(* CODESYS project 4D_Handling_Demo_Seti.project

Project tree, tasks and I/O mapping:
  Device : CPX-CEC-M1-V3, Festo AG & Co. KG, order no. 3472765, version 3.5.7.25
      unmapped channels: Rotary switch
    application Application
      libraries: Standard, * (System); CAA CiA 405, 3.5.7.0 (CAA Technical Workgroup); Festo_Motion_FHPP_3, 3.5.5.0 (Festo AG & Co. KG)
      task MainTask (cyclic, interval t#20ms, priority 20) calls Main_PRG
      program Main_PRG [ST]
      PO3_Axis/
        AxisX/
          program PrgAxisXCallPrg [ST]
      program Motion_PRG [ST]
      program FHPP [CFC]
      global variables Global
      visualisation Visualization
    PLC_Diagnosis : PLC-Diagnosis, Festo AG & Co. KG, version 3.5.4.1
    CPX_System : CPX_System, Festo AG & Co. KG, order no. 3472765, version 1.200
      _8DI_8DO : 8DI/8DO, Festo AG & Co. KG, order no. 526257, version 1.200
          unmapped channels: Input 0, Output 0
      _8DI_8DO_1 : 8DI/8DO, Festo AG & Co. KG, order no. 526257, version 1.200
          settings:  = 0;  = 1;  = 1;  = 1;  = 1;  = 0;  = 1;  = 1;  = 0;  = 0;  = 0;  = 0;  = 0;  = 0;  = 0;  = 0;  = 0;  = 0;  = 0;  = 0;  = 0;  = 0;  = 0;  = 0;  = 0;  = 0;  = 0;  = 0;  = 0;  = 0;  = 0;  = 0;  = 0;  = 0;  = 0;  = 0;  = 0;  = 0;  = 0;  = 0;
             = 0;  = 0;  = 0;  = 0;  = 0;  = 0;  = 0;  = 0;  = 0;  = 0;  = 0;  = 0;  = 0;  = 0;  = 0;  = 0;  = 0;  = 0;  = 0;  = 0;  = 0;  = 0;  = 0;  = 0;  = 0;  = 0;  = 0;  = 0;  = 0;  = 0;  = 0;  = 0;  = 0;  = 0;  = 0;  = 0;  = 0;  = 0;  = 0;  = 0;
             = 576751027668385792;  = 'PI%i.0.0.1=1';  = 'PI%i.0.1.1=1';  = 'PI%i.0.2.1=1';  = 'PI%i.1.0.1=1';  = 'PI%i.1.1.1=0';  = 'PI%i.1.4.2=1';  = 'PI%i.1.6.2=1';  = 'PI%i.6.0.1=0';  = 'PI%i.6.1.1=0';  = 'PI%i.6.2.1=0';  = 'PI%i.6.3.1=0';  = 'PI%i.6.4.1=0';  = 'PI%i.6.5.1=0';  = 'PI%i.6.6.1=0';  = 'PI%i.6.7.1=0';  = dd1ef60a;  = 6
          unmapped channels: Input 0, Output 0
      CEC_M1_V3 : CEC-M1-V3, Festo AG & Co. KG, order no. 3472765, version 1.200
          settings:  = 0;  = 196272706293248;  = 352692416;  = 16777215;  = 0;  = 13959209;  = 1f4c82b2;  = 5
    SoftMotion General Axis Pool
    CAN : CANbus, 3S - Smart Software Solutions GmbH, version 3.5.7.0
        settings: Baudrate = 1000
      CANopen : CANopen_Manager, 3S - Smart Software Solutions GmbH, version 3.5.7.20
          settings: Sync CycleTime in Microseconds = 8000; Synchronous Window Length = 0; Enable Heartbeat generation = FALSE; Factory Settings Default = FALSE; Expert Settings Default = TRUE; ConfigVersion = 50659584
        U3 : CMMP-AS-C5-3A-M0 (FHPP), Festo AG & Co. KG, order no. 1622902, version 0.262146.CMMP_AS_C5_3A_M0_FHPP.2.8
            settings: General Options.Reset Node = FALSE; NODEIDSAVED = 3; SDO Timeout = 1000000; PDO_Autoconfig = FALSE; EXPERTSETTINGS = TRUE; Emergency-General Parameters.Emergency COBID = 16#00000083; PDO 16#1400.COBID = 16#00000203; PDO 16#1401.COBID = 16#00000303; PDO 16#1402.COBID = 16#00000403; PDO 16#1403.COBID = 16#00000503; PDO 16#1800.COBID = 16#00000183; PDO 16#1800.Event Timer = 0; PDO 16#1801.COBID = 16#00000283; PDO 16#1801.Event Timer = 0; PDO 16#1802.COBID = 16#00000383; PDO 16#1802.Event Timer = 0; PDO 16#1803.COBID = 16#00000483; PDO 16#1803.Event Timer = 0; CCON.Subindex = 16#00; CPOS.Subindex = 16#00; REC_NR/CDIR.Subindex = 16#00; RES/DEM_VAL1/PARA1.Subindex = 16#00; RES/DEM_VAL2/PARA2.Subindex = 16#00; RES.Subindex = 16#00; SUBINDEX.Subindex = 16#00; REQCODE_PNU.Subindex = 16#00; PARAVAL.Subindex = 16#00; FHPP+_O_Byte01.Subindex = 16#00; FHPP+_O_Byte02.Subindex = 16#00; FHPP+_O_Byte03.Subindex = 16#00; FHPP+_O_Byte04.Subindex = 16#00; FHPP+_O_Byte05.Subindex = 16#00; FHPP+_O_Byte06.Subindex = 16#00; FHPP+_O_Byte07.Subindex = 16#00; FHPP+_O_Byte08.Subindex = 16#00; FHPP+_O_Byte09.Subindex = 16#00; FHPP+_O_Byte10.Subindex = 16#00; FHPP+_O_Byte11.Subindex = 16#00; FHPP+_O_Byte12.Subindex = 16#00; FHPP+_O_Byte13.Subindex = 16#00;
              FHPP+_O_Byte14.Subindex = 16#00; FHPP+_O_Byte15.Subindex = 16#00; FHPP+_O_Byte16.Subindex = 16#00; SCON.Subindex = 16#00; SPOS.Subindex = 16#00; REC_NR/SDIR.Subindex = 16#00; RSB/ACT_VAL1.Subindex = 16#00; ACT_POS/ACT_VAL2.Subindex = 16#00; RES.Subindex = 16#00; SUBINDEX.Subindex = 16#00; RESPCODE_PNU.Subindex = 16#00; PARAVAL.Subindex = 16#00; FHPP+_I_Byte01.Subindex = 16#00; FHPP+_I_Byte02.Subindex = 16#00; FHPP+_I_Byte03.Subindex = 16#00; FHPP+_I_Byte04.Subindex = 16#00; FHPP+_I_Byte05.Subindex = 16#00; FHPP+_I_Byte06.Subindex = 16#00; FHPP+_I_Byte07.Subindex = 16#00; FHPP+_I_Byte08.Subindex = 16#00; FHPP+_I_Byte09.Subindex = 16#00; FHPP+_I_Byte10.Subindex = 16#00; FHPP+_I_Byte11.Subindex = 16#00; FHPP+_I_Byte12.Subindex = 16#00; FHPP+_I_Byte13.Subindex = 16#00; FHPP+_I_Byte14.Subindex = 16#00; FHPP+_I_Byte15.Subindex = 16#00; FHPP+_I_Byte16.Subindex = 16#00; SDO List.Disable TIME.Index = 16#1012; SDO List.Disable TIME.Subindex = 16#00; SDO List.Disable TIME.Value = 16#00000100; SDO List.Disable TIME.Size = 32; SDO List.Disable TIME.AbortIfError = FALSE; SDO List.Disable TIME.JumpToLine = FALSE; SDO List.Disable TIME.Line = 0; SDO List.Set Guardtime.Index = 16#100C; SDO List.Set Guardtime.Subindex = 16#00; SDO List.Set Guardtime.Value = 16#00000000; SDO List.Set Guardtime.Size = 16; SDO List.Set Guardtime.AbortIfError = FALSE;
              SDO List.Set Guardtime.JumpToLine = FALSE; SDO List.Set Guardtime.Line = 0; SDO List.Set Lifetime.Index = 16#100D; SDO List.Set Lifetime.Subindex = 16#00; SDO List.Set Lifetime.Value = 16#00000000; SDO List.Set Lifetime.Size = 8; SDO List.Set Lifetime.AbortIfError = FALSE; SDO List.Set Lifetime.JumpToLine = FALSE; SDO List.Set Lifetime.Line = 0; SDO List.Disable Emcy CobID.Index = 16#1014; SDO List.Disable Emcy CobID.Subindex = 16#00; SDO List.Disable Emcy CobID.Value = 16#80000083; SDO List.Disable Emcy CobID.Size = 32; SDO List.Disable Emcy CobID.AbortIfError = FALSE; SDO List.Disable Emcy CobID.JumpToLine = FALSE; SDO List.Disable Emcy CobID.Line = 0; SDO List.Set Emcy CobID.Index = 16#1014; SDO List.Set Emcy CobID.Subindex = 16#00; SDO List.Set Emcy CobID.Value = 16#00000083; SDO List.Set Emcy CobID.Size = 32; SDO List.Set Emcy CobID.AbortIfError = FALSE; SDO List.Set Emcy CobID.JumpToLine = FALSE; SDO List.Set Emcy CobID.Line = 0; SDO List.Set Heartbeat Consumer.Index = 16#1016; SDO List.Set Heartbeat Consumer.Subindex = 16#01; SDO List.Set Heartbeat Consumer.Value = 0; SDO List.Set Heartbeat Consumer.Size = 32; SDO List.Set Heartbeat Consumer.AbortIfError = FALSE; SDO List.Set Heartbeat Consumer.JumpToLine = FALSE; SDO List.Set Heartbeat Consumer.Line = 0; SDO List.Set Heartbeat Producer.Index = 16#1017; SDO List.Set Heartbeat Producer.Subindex = 16#00; SDO List.Set Heartbeat Producer.Value = 16#00000000; SDO List.Set Heartbeat Producer.Size = 16; SDO List.Set Heartbeat Producer.AbortIfError = FALSE; SDO List.Set Heartbeat Producer.JumpToLine = FALSE; SDO List.Set Heartbeat Producer.Line = 0; SDO List.Disable PDO.Index = 16#1400; SDO List.Disable PDO.Subindex = 16#01; SDO List.Disable PDO.Value = 16#80000203;
              SDO List.Disable PDO.Size = 32; SDO List.Disable PDO.AbortIfError = FALSE; SDO List.Disable PDO.JumpToLine = FALSE; SDO List.Disable PDO.Line = 0; SDO List.Set transmission type.Index = 16#1400; SDO List.Set transmission type.Subindex = 16#02; SDO List.Set transmission type.Value = 16#FF; SDO List.Set transmission type.Size = 8; SDO List.Set transmission type.AbortIfError = FALSE; SDO List.Set transmission type.JumpToLine = FALSE; SDO List.Set transmission type.Line = 0; SDO List.Set and enable COB-ID.Index = 16#1400; SDO List.Set and enable COB-ID.Subindex = 16#01; SDO List.Set and enable COB-ID.Value = 16#00000203; SDO List.Set and enable COB-ID.Size = 32; SDO List.Set and enable COB-ID.AbortIfError = FALSE; SDO List.Set and enable COB-ID.JumpToLine = FALSE; SDO List.Set and enable COB-ID.Line = 0; SDO List.Disable PDO.Index = 16#1401; SDO List.Disable PDO.Subindex = 16#01; SDO List.Disable PDO.Value = 16#80000303; SDO List.Disable PDO.Size = 32; SDO List.Disable PDO.AbortIfError = FALSE; SDO List.Disable PDO.JumpToLine = FALSE; SDO List.Disable PDO.Line = 0; SDO List.Set transmission type.Index = 16#1401; SDO List.Set transmission type.Subindex = 16#02; SDO List.Set transmission type.Value = 16#FF; SDO List.Set transmission type.Size = 8; SDO List.Set transmission type.AbortIfError = FALSE; SDO List.Set transmission type.JumpToLine = FALSE; SDO List.Set transmission type.Line = 0; SDO List.Set and enable COB-ID.Index = 16#1401; SDO List.Set and enable COB-ID.Subindex = 16#01; SDO List.Set and enable COB-ID.Value = 16#00000303; SDO List.Set and enable COB-ID.Size = 32; SDO List.Set and enable COB-ID.AbortIfError = FALSE; SDO List.Set and enable COB-ID.JumpToLine = FALSE; SDO List.Set and enable COB-ID.Line = 0; SDO List.Disable PDO.Index = 16#1402;
              SDO List.Disable PDO.Subindex = 16#01; SDO List.Disable PDO.Value = 16#80000403; SDO List.Disable PDO.Size = 32; SDO List.Disable PDO.AbortIfError = FALSE; SDO List.Disable PDO.JumpToLine = FALSE; SDO List.Disable PDO.Line = 0; SDO List.Set transmission type.Index = 16#1402; SDO List.Set transmission type.Subindex = 16#02; SDO List.Set transmission type.Value = 16#FF; SDO List.Set transmission type.Size = 8; SDO List.Set transmission type.AbortIfError = FALSE; SDO List.Set transmission type.JumpToLine = FALSE; SDO List.Set transmission type.Line = 0; SDO List.Clear pdo mapping.Index = 16#1602; SDO List.Clear pdo mapping.Subindex = 16#00; SDO List.Clear pdo mapping.Value = 16#0; SDO List.Clear pdo mapping.Size = 8; SDO List.Clear pdo mapping.AbortIfError = FALSE; SDO List.Clear pdo mapping.JumpToLine = FALSE; SDO List.Clear pdo mapping.Line = 0; SDO List.Set Mapping.Index = 16#1602; SDO List.Set Mapping.Subindex = 16#01; SDO List.Set Mapping.Value = 16#31010008; SDO List.Set Mapping.Size = 32; SDO List.Set Mapping.AbortIfError = FALSE; SDO List.Set Mapping.JumpToLine = FALSE; SDO List.Set Mapping.Line = 0; SDO List.Set Mapping.Index = 16#1602; SDO List.Set Mapping.Subindex = 16#02; SDO List.Set Mapping.Value = 16#31020008; SDO List.Set Mapping.Size = 32; SDO List.Set Mapping.AbortIfError = FALSE; SDO List.Set Mapping.JumpToLine = FALSE; SDO List.Set Mapping.Line = 0; SDO List.Set Mapping.Index = 16#1602; SDO List.Set Mapping.Subindex = 16#03; SDO List.Set Mapping.Value = 16#31030008; SDO List.Set Mapping.Size = 32; SDO List.Set Mapping.AbortIfError = FALSE; SDO List.Set Mapping.JumpToLine = FALSE;
              SDO List.Set Mapping.Line = 0; SDO List.Set Mapping.Index = 16#1602; SDO List.Set Mapping.Subindex = 16#04; SDO List.Set Mapping.Value = 16#31040008; SDO List.Set Mapping.Size = 32; SDO List.Set Mapping.AbortIfError = FALSE; SDO List.Set Mapping.JumpToLine = FALSE; SDO List.Set Mapping.Line = 0; SDO List.Set Mapping.Index = 16#1602; SDO List.Set Mapping.Subindex = 16#05; SDO List.Set Mapping.Value = 16#31050008; SDO List.Set Mapping.Size = 32; SDO List.Set Mapping.AbortIfError = FALSE; SDO List.Set Mapping.JumpToLine = FALSE; SDO List.Set Mapping.Line = 0; SDO List.Set Mapping.Index = 16#1602; SDO List.Set Mapping.Subindex = 16#06; SDO List.Set Mapping.Value = 16#31060008; SDO List.Set Mapping.Size = 32; SDO List.Set Mapping.AbortIfError = FALSE; SDO List.Set Mapping.JumpToLine = FALSE; SDO List.Set Mapping.Line = 0; SDO List.Set Mapping.Index = 16#1602; SDO List.Set Mapping.Subindex = 16#07; SDO List.Set Mapping.Value = 16#31070008; SDO List.Set Mapping.Size = 32; SDO List.Set Mapping.AbortIfError = FALSE; SDO List.Set Mapping.JumpToLine = FALSE; SDO List.Set Mapping.Line = 0; SDO List.Set Mapping.Index = 16#1602; SDO List.Set Mapping.Subindex = 16#08; SDO List.Set Mapping.Value = 16#31080008; SDO List.Set Mapping.Size = 32; SDO List.Set Mapping.AbortIfError = FALSE; SDO List.Set Mapping.JumpToLine = FALSE; SDO List.Set Mapping.Line = 0; SDO List.Set number of mappings.Index = 16#1602; SDO List.Set number of mappings.Subindex = 16#00; SDO List.Set number of mappings.Value = 16#08; SDO List.Set number of mappings.Size = 8;
              SDO List.Set number of mappings.AbortIfError = FALSE; SDO List.Set number of mappings.JumpToLine = FALSE; SDO List.Set number of mappings.Line = 0; SDO List.Set and enable COB-ID.Index = 16#1402; SDO List.Set and enable COB-ID.Subindex = 16#01; SDO List.Set and enable COB-ID.Value = 16#00000403; SDO List.Set and enable COB-ID.Size = 32; SDO List.Set and enable COB-ID.AbortIfError = FALSE; SDO List.Set and enable COB-ID.JumpToLine = FALSE; SDO List.Set and enable COB-ID.Line = 0; SDO List.Disable PDO.Index = 16#1403; SDO List.Disable PDO.Subindex = 16#01; SDO List.Disable PDO.Value = 16#80000503; SDO List.Disable PDO.Size = 32; SDO List.Disable PDO.AbortIfError = FALSE; SDO List.Disable PDO.JumpToLine = FALSE; SDO List.Disable PDO.Line = 0; SDO List.Set transmission type.Index = 16#1403; SDO List.Set transmission type.Subindex = 16#02; SDO List.Set transmission type.Value = 16#FF; SDO List.Set transmission type.Size = 8; SDO List.Set transmission type.AbortIfError = FALSE; SDO List.Set transmission type.JumpToLine = FALSE; SDO List.Set transmission type.Line = 0; SDO List.Clear pdo mapping.Index = 16#1603; SDO List.Clear pdo mapping.Subindex = 16#00; SDO List.Clear pdo mapping.Value = 16#0; SDO List.Clear pdo mapping.Size = 8; SDO List.Clear pdo mapping.AbortIfError = FALSE; SDO List.Clear pdo mapping.JumpToLine = FALSE; SDO List.Clear pdo mapping.Line = 0; SDO List.Set Mapping.Index = 16#1603; SDO List.Set Mapping.Subindex = 16#01; SDO List.Set Mapping.Value = 16#31090008; SDO List.Set Mapping.Size = 32; SDO List.Set Mapping.AbortIfError = FALSE; SDO List.Set Mapping.JumpToLine = FALSE; SDO List.Set Mapping.Line = 0; SDO List.Set Mapping.Index = 16#1603; SDO List.Set Mapping.Subindex = 16#02;
              SDO List.Set Mapping.Value = 16#31100008; SDO List.Set Mapping.Size = 32; SDO List.Set Mapping.AbortIfError = FALSE; SDO List.Set Mapping.JumpToLine = FALSE; SDO List.Set Mapping.Line = 0; SDO List.Set Mapping.Index = 16#1603; SDO List.Set Mapping.Subindex = 16#03; SDO List.Set Mapping.Value = 16#31110008; SDO List.Set Mapping.Size = 32; SDO List.Set Mapping.AbortIfError = FALSE; SDO List.Set Mapping.JumpToLine = FALSE; SDO List.Set Mapping.Line = 0; SDO List.Set Mapping.Index = 16#1603; SDO List.Set Mapping.Subindex = 16#04; SDO List.Set Mapping.Value = 16#31120008; SDO List.Set Mapping.Size = 32; SDO List.Set Mapping.AbortIfError = FALSE; SDO List.Set Mapping.JumpToLine = FALSE; SDO List.Set Mapping.Line = 0; SDO List.Set Mapping.Index = 16#1603; SDO List.Set Mapping.Subindex = 16#05; SDO List.Set Mapping.Value = 16#31130008; SDO List.Set Mapping.Size = 32; SDO List.Set Mapping.AbortIfError = FALSE; SDO List.Set Mapping.JumpToLine = FALSE; SDO List.Set Mapping.Line = 0; SDO List.Set Mapping.Index = 16#1603; SDO List.Set Mapping.Subindex = 16#06; SDO List.Set Mapping.Value = 16#31140008; SDO List.Set Mapping.Size = 32; SDO List.Set Mapping.AbortIfError = FALSE; SDO List.Set Mapping.JumpToLine = FALSE; SDO List.Set Mapping.Line = 0; SDO List.Set Mapping.Index = 16#1603; SDO List.Set Mapping.Subindex = 16#07; SDO List.Set Mapping.Value = 16#31150008; SDO List.Set Mapping.Size = 32; SDO List.Set Mapping.AbortIfError = FALSE; SDO List.Set Mapping.JumpToLine = FALSE; SDO List.Set Mapping.Line = 0;
              SDO List.Set Mapping.Index = 16#1603; SDO List.Set Mapping.Subindex = 16#08; SDO List.Set Mapping.Value = 16#31160008; SDO List.Set Mapping.Size = 32; SDO List.Set Mapping.AbortIfError = FALSE; SDO List.Set Mapping.JumpToLine = FALSE; SDO List.Set Mapping.Line = 0; SDO List.Set number of mappings.Index = 16#1603; SDO List.Set number of mappings.Subindex = 16#00; SDO List.Set number of mappings.Value = 16#08; SDO List.Set number of mappings.Size = 8; SDO List.Set number of mappings.AbortIfError = FALSE; SDO List.Set number of mappings.JumpToLine = FALSE; SDO List.Set number of mappings.Line = 0; SDO List.Set and enable COB-ID.Index = 16#1403; SDO List.Set and enable COB-ID.Subindex = 16#01; SDO List.Set and enable COB-ID.Value = 16#00000503; SDO List.Set and enable COB-ID.Size = 32; SDO List.Set and enable COB-ID.AbortIfError = FALSE; SDO List.Set and enable COB-ID.JumpToLine = FALSE; SDO List.Set and enable COB-ID.Line = 0; SDO List.Disable PDO.Index = 16#1800; SDO List.Disable PDO.Subindex = 16#01; SDO List.Disable PDO.Value = 16#80000183; SDO List.Disable PDO.Size = 32; SDO List.Disable PDO.AbortIfError = FALSE; SDO List.Disable PDO.JumpToLine = FALSE; SDO List.Disable PDO.Line = 0; SDO List.Set transmission type.Index = 16#1800; SDO List.Set transmission type.Subindex = 16#02; SDO List.Set transmission type.Value = 16#FF; SDO List.Set transmission type.Size = 8; SDO List.Set transmission type.AbortIfError = FALSE; SDO List.Set transmission type.JumpToLine = FALSE; SDO List.Set transmission type.Line = 0; SDO List.Set inhibit time.Index = 16#1800; SDO List.Set inhibit time.Subindex = 16#03; SDO List.Set inhibit time.Value = 16#0000; SDO List.Set inhibit time.Size = 16; SDO List.Set inhibit time.AbortIfError = FALSE;
              SDO List.Set inhibit time.JumpToLine = FALSE; SDO List.Set inhibit time.Line = 0; SDO List.Set and enable COB-ID.Index = 16#1800; SDO List.Set and enable COB-ID.Subindex = 16#01; SDO List.Set and enable COB-ID.Value = 16#00000183; SDO List.Set and enable COB-ID.Size = 32; SDO List.Set and enable COB-ID.AbortIfError = FALSE; SDO List.Set and enable COB-ID.JumpToLine = FALSE; SDO List.Set and enable COB-ID.Line = 0; SDO List.Disable PDO.Index = 16#1801; SDO List.Disable PDO.Subindex = 16#01; SDO List.Disable PDO.Value = 16#80000283; SDO List.Disable PDO.Size = 32; SDO List.Disable PDO.AbortIfError = FALSE; SDO List.Disable PDO.JumpToLine = FALSE; SDO List.Disable PDO.Line = 0; SDO List.Set transmission type.Index = 16#1801; SDO List.Set transmission type.Subindex = 16#02; SDO List.Set transmission type.Value = 16#FF; SDO List.Set transmission type.Size = 8; SDO List.Set transmission type.AbortIfError = FALSE; SDO List.Set transmission type.JumpToLine = FALSE; SDO List.Set transmission type.Line = 0; SDO List.Set inhibit time.Index = 16#1801; SDO List.Set inhibit time.Subindex = 16#03; SDO List.Set inhibit time.Value = 16#0000; SDO List.Set inhibit time.Size = 16; SDO List.Set inhibit time.AbortIfError = FALSE; SDO List.Set inhibit time.JumpToLine = FALSE; SDO List.Set inhibit time.Line = 0; SDO List.Set and enable COB-ID.Index = 16#1801; SDO List.Set and enable COB-ID.Subindex = 16#01; SDO List.Set and enable COB-ID.Value = 16#00000283; SDO List.Set and enable COB-ID.Size = 32; SDO List.Set and enable COB-ID.AbortIfError = FALSE; SDO List.Set and enable COB-ID.JumpToLine = FALSE; SDO List.Set and enable COB-ID.Line = 0; SDO List.Disable PDO.Index = 16#1802; SDO List.Disable PDO.Subindex = 16#01; SDO List.Disable PDO.Value = 16#80000383;
              SDO List.Disable PDO.Size = 32; SDO List.Disable PDO.AbortIfError = FALSE; SDO List.Disable PDO.JumpToLine = FALSE; SDO List.Disable PDO.Line = 0; SDO List.Set transmission type.Index = 16#1802; SDO List.Set transmission type.Subindex = 16#02; SDO List.Set transmission type.Value = 16#FF; SDO List.Set transmission type.Size = 8; SDO List.Set transmission type.AbortIfError = FALSE; SDO List.Set transmission type.JumpToLine = FALSE; SDO List.Set transmission type.Line = 0; SDO List.Set inhibit time.Index = 16#1802; SDO List.Set inhibit time.Subindex = 16#03; SDO List.Set inhibit time.Value = 16#0000; SDO List.Set inhibit time.Size = 16; SDO List.Set inhibit time.AbortIfError = FALSE; SDO List.Set inhibit time.JumpToLine = FALSE; SDO List.Set inhibit time.Line = 0; SDO List.Clear pdo mapping.Index = 16#1A02; SDO List.Clear pdo mapping.Subindex = 16#00; SDO List.Clear pdo mapping.Value = 16#0; SDO List.Clear pdo mapping.Size = 8; SDO List.Clear pdo mapping.AbortIfError = FALSE; SDO List.Clear pdo mapping.JumpToLine = FALSE; SDO List.Clear pdo mapping.Line = 0; SDO List.Set Mapping.Index = 16#1A02; SDO List.Set Mapping.Subindex = 16#01; SDO List.Set Mapping.Value = 16#32010008; SDO List.Set Mapping.Size = 32; SDO List.Set Mapping.AbortIfError = FALSE; SDO List.Set Mapping.JumpToLine = FALSE; SDO List.Set Mapping.Line = 0; SDO List.Set Mapping.Index = 16#1A02; SDO List.Set Mapping.Subindex = 16#02; SDO List.Set Mapping.Value = 16#32020008; SDO List.Set Mapping.Size = 32; SDO List.Set Mapping.AbortIfError = FALSE; SDO List.Set Mapping.JumpToLine = FALSE; SDO List.Set Mapping.Line = 0; SDO List.Set Mapping.Index = 16#1A02;
              SDO List.Set Mapping.Subindex = 16#03; SDO List.Set Mapping.Value = 16#32030008; SDO List.Set Mapping.Size = 32; SDO List.Set Mapping.AbortIfError = FALSE; SDO List.Set Mapping.JumpToLine = FALSE; SDO List.Set Mapping.Line = 0; SDO List.Set Mapping.Index = 16#1A02; SDO List.Set Mapping.Subindex = 16#04; SDO List.Set Mapping.Value = 16#32040008; SDO List.Set Mapping.Size = 32; SDO List.Set Mapping.AbortIfError = FALSE; SDO List.Set Mapping.JumpToLine = FALSE; SDO List.Set Mapping.Line = 0; SDO List.Set Mapping.Index = 16#1A02; SDO List.Set Mapping.Subindex = 16#05; SDO List.Set Mapping.Value = 16#32050008; SDO List.Set Mapping.Size = 32; SDO List.Set Mapping.AbortIfError = FALSE; SDO List.Set Mapping.JumpToLine = FALSE; SDO List.Set Mapping.Line = 0; SDO List.Set Mapping.Index = 16#1A02; SDO List.Set Mapping.Subindex = 16#06; SDO List.Set Mapping.Value = 16#32060008; SDO List.Set Mapping.Size = 32; SDO List.Set Mapping.AbortIfError = FALSE; SDO List.Set Mapping.JumpToLine = FALSE; SDO List.Set Mapping.Line = 0; SDO List.Set Mapping.Index = 16#1A02; SDO List.Set Mapping.Subindex = 16#07; SDO List.Set Mapping.Value = 16#32070008; SDO List.Set Mapping.Size = 32; SDO List.Set Mapping.AbortIfError = FALSE; SDO List.Set Mapping.JumpToLine = FALSE; SDO List.Set Mapping.Line = 0; SDO List.Set Mapping.Index = 16#1A02; SDO List.Set Mapping.Subindex = 16#08; SDO List.Set Mapping.Value = 16#32080008; SDO List.Set Mapping.Size = 32; SDO List.Set Mapping.AbortIfError = FALSE; SDO List.Set Mapping.JumpToLine = FALSE;
              SDO List.Set Mapping.Line = 0; SDO List.Set number of mappings.Index = 16#1A02; SDO List.Set number of mappings.Subindex = 16#00; SDO List.Set number of mappings.Value = 16#08; SDO List.Set number of mappings.Size = 8; SDO List.Set number of mappings.AbortIfError = FALSE; SDO List.Set number of mappings.JumpToLine = FALSE; SDO List.Set number of mappings.Line = 0; SDO List.Set and enable COB-ID.Index = 16#1802; SDO List.Set and enable COB-ID.Subindex = 16#01; SDO List.Set and enable COB-ID.Value = 16#00000383; SDO List.Set and enable COB-ID.Size = 32; SDO List.Set and enable COB-ID.AbortIfError = FALSE; SDO List.Set and enable COB-ID.JumpToLine = FALSE; SDO List.Set and enable COB-ID.Line = 0; SDO List.Disable PDO.Index = 16#1803; SDO List.Disable PDO.Subindex = 16#01; SDO List.Disable PDO.Value = 16#80000483; SDO List.Disable PDO.Size = 32; SDO List.Disable PDO.AbortIfError = FALSE; SDO List.Disable PDO.JumpToLine = FALSE; SDO List.Disable PDO.Line = 0; SDO List.Set transmission type.Index = 16#1803; SDO List.Set transmission type.Subindex = 16#02; SDO List.Set transmission type.Value = 16#FF; SDO List.Set transmission type.Size = 8; SDO List.Set transmission type.AbortIfError = FALSE; SDO List.Set transmission type.JumpToLine = FALSE; SDO List.Set transmission type.Line = 0; SDO List.Set inhibit time.Index = 16#1803; SDO List.Set inhibit time.Subindex = 16#03; SDO List.Set inhibit time.Value = 16#0000; SDO List.Set inhibit time.Size = 16; SDO List.Set inhibit time.AbortIfError = FALSE; SDO List.Set inhibit time.JumpToLine = FALSE; SDO List.Set inhibit time.Line = 0; SDO List.Clear pdo mapping.Index = 16#1A03; SDO List.Clear pdo mapping.Subindex = 16#00; SDO List.Clear pdo mapping.Value = 16#0; SDO List.Clear pdo mapping.Size = 8;
              SDO List.Clear pdo mapping.AbortIfError = FALSE; SDO List.Clear pdo mapping.JumpToLine = FALSE; SDO List.Clear pdo mapping.Line = 0; SDO List.Set Mapping.Index = 16#1A03; SDO List.Set Mapping.Subindex = 16#01; SDO List.Set Mapping.Value = 16#32090008; SDO List.Set Mapping.Size = 32; SDO List.Set Mapping.AbortIfError = FALSE; SDO List.Set Mapping.JumpToLine = FALSE; SDO List.Set Mapping.Line = 0; SDO List.Set Mapping.Index = 16#1A03; SDO List.Set Mapping.Subindex = 16#02; SDO List.Set Mapping.Value = 16#32100008; SDO List.Set Mapping.Size = 32; SDO List.Set Mapping.AbortIfError = FALSE; SDO List.Set Mapping.JumpToLine = FALSE; SDO List.Set Mapping.Line = 0; SDO List.Set Mapping.Index = 16#1A03; SDO List.Set Mapping.Subindex = 16#03; SDO List.Set Mapping.Value = 16#32110008; SDO List.Set Mapping.Size = 32; SDO List.Set Mapping.AbortIfError = FALSE; SDO List.Set Mapping.JumpToLine = FALSE; SDO List.Set Mapping.Line = 0; SDO List.Set Mapping.Index = 16#1A03; SDO List.Set Mapping.Subindex = 16#04; SDO List.Set Mapping.Value = 16#32120008; SDO List.Set Mapping.Size = 32; SDO List.Set Mapping.AbortIfError = FALSE; SDO List.Set Mapping.JumpToLine = FALSE; SDO List.Set Mapping.Line = 0; SDO List.Set Mapping.Index = 16#1A03; SDO List.Set Mapping.Subindex = 16#05; SDO List.Set Mapping.Value = 16#32130008; SDO List.Set Mapping.Size = 32; SDO List.Set Mapping.AbortIfError = FALSE; SDO List.Set Mapping.JumpToLine = FALSE; SDO List.Set Mapping.Line = 0; SDO List.Set Mapping.Index = 16#1A03; SDO List.Set Mapping.Subindex = 16#06;
              SDO List.Set Mapping.Value = 16#32140008; SDO List.Set Mapping.Size = 32; SDO List.Set Mapping.AbortIfError = FALSE; SDO List.Set Mapping.JumpToLine = FALSE; SDO List.Set Mapping.Line = 0; SDO List.Set Mapping.Index = 16#1A03; SDO List.Set Mapping.Subindex = 16#07; SDO List.Set Mapping.Value = 16#32150008; SDO List.Set Mapping.Size = 32; SDO List.Set Mapping.AbortIfError = FALSE; SDO List.Set Mapping.JumpToLine = FALSE; SDO List.Set Mapping.Line = 0; SDO List.Set Mapping.Index = 16#1A03; SDO List.Set Mapping.Subindex = 16#08; SDO List.Set Mapping.Value = 16#32160008; SDO List.Set Mapping.Size = 32; SDO List.Set Mapping.AbortIfError = FALSE; SDO List.Set Mapping.JumpToLine = FALSE; SDO List.Set Mapping.Line = 0; SDO List.Set number of mappings.Index = 16#1A03; SDO List.Set number of mappings.Subindex = 16#00; SDO List.Set number of mappings.Value = 16#08; SDO List.Set number of mappings.Size = 8; SDO List.Set number of mappings.AbortIfError = FALSE; SDO List.Set number of mappings.JumpToLine = FALSE; SDO List.Set number of mappings.Line = 0; SDO List.Set and enable COB-ID.Index = 16#1803; SDO List.Set and enable COB-ID.Subindex = 16#01; SDO List.Set and enable COB-ID.Value = 16#00000483; SDO List.Set and enable COB-ID.Size = 32; SDO List.Set and enable COB-ID.AbortIfError = FALSE; SDO List.Set and enable COB-ID.JumpToLine = FALSE; SDO List.Set and enable COB-ID.Line = 0; ConfigVersion = 50659584
            unmapped channels: CCON, CPOS, REC_NR/CDIR, RES/DEM_VAL1/PARA1, RES/DEM_VAL2/PARA2, RES, SUBINDEX, REQCODE_PNU, PARAVAL, FHPP+_O_Byte01, FHPP+_O_Byte02, FHPP+_O_Byte03, FHPP+_O_Byte04, FHPP+_O_Byte05, FHPP+_O_Byte06, FHPP+_O_Byte07, FHPP+_O_Byte08, FHPP+_O_Byte09, FHPP+_O_Byte10, FHPP+_O_Byte11, FHPP+_O_Byte12, FHPP+_O_Byte13, FHPP+_O_Byte14, FHPP+_O_Byte15, FHPP+_O_Byte16, SCON, SPOS, REC_NR/SDIR, RSB/ACT_VAL1, ACT_POS/ACT_VAL2, RES, SUBINDEX, RESPCODE_PNU, PARAVAL, FHPP+_I_Byte01, FHPP+_I_Byte02, FHPP+_I_Byte03, FHPP+_I_Byte04, FHPP+_I_Byte05, FHPP+_I_Byte06,
              FHPP+_I_Byte07, FHPP+_I_Byte08, FHPP+_I_Byte09, FHPP+_I_Byte10, FHPP+_I_Byte11, FHPP+_I_Byte12, FHPP+_I_Byte13, FHPP+_I_Byte14, FHPP+_I_Byte15, FHPP+_I_Byte16
        U1 : CMMP-AS-C5-3A-M0 (FHPP), Festo AG & Co. KG, order no. 1622902, version 0.262146.CMMP_AS_C5_3A_M0_FHPP.2.8
            settings: General Options.Reset Node = FALSE; NODEIDSAVED = 1; SDO Timeout = 1000000; EXPERTSETTINGS = TRUE; PDO 16#1400.COBID = 16#00000201; PDO 16#1401.COBID = 16#00000301; PDO 16#1402.COBID = 16#00000401; PDO 16#1403.COBID = 16#00000501; PDO 16#1800.COBID = 16#00000181; PDO 16#1800.Event Timer = 0; PDO 16#1801.COBID = 16#00000281; PDO 16#1801.Event Timer = 0; PDO 16#1802.COBID = 16#00000381; PDO 16#1802.Event Timer = 0; PDO 16#1803.COBID = 16#00000481; PDO 16#1803.Event Timer = 0; CCON.Subindex = 16#00; CPOS.Subindex = 16#00; REC_NR/CDIR.Subindex = 16#00; RES/DEM_VAL1/PARA1.Subindex = 16#00; RES/DEM_VAL2/PARA2.Subindex = 16#00; RES.Subindex = 16#00; SUBINDEX.Subindex = 16#00; REQCODE_PNU.Subindex = 16#00; PARAVAL.Subindex = 16#00; FHPP+_O_Byte01.Subindex = 16#00; FHPP+_O_Byte02.Subindex = 16#00; FHPP+_O_Byte03.Subindex = 16#00; FHPP+_O_Byte04.Subindex = 16#00; FHPP+_O_Byte05.Subindex = 16#00; FHPP+_O_Byte06.Subindex = 16#00; FHPP+_O_Byte07.Subindex = 16#00; FHPP+_O_Byte08.Subindex = 16#00; FHPP+_O_Byte09.Subindex = 16#00; FHPP+_O_Byte10.Subindex = 16#00; FHPP+_O_Byte11.Subindex = 16#00; FHPP+_O_Byte12.Subindex = 16#00; FHPP+_O_Byte13.Subindex = 16#00; FHPP+_O_Byte14.Subindex = 16#00; FHPP+_O_Byte15.Subindex = 16#00;
              FHPP+_O_Byte16.Subindex = 16#00; SCON.Subindex = 16#00; SPOS.Subindex = 16#00; REC_NR/SDIR.Subindex = 16#00; RSB/ACT_VAL1.Subindex = 16#00; ACT_POS/ACT_VAL2.Subindex = 16#00; RES.Subindex = 16#00; SUBINDEX.Subindex = 16#00; RESPCODE_PNU.Subindex = 16#00; PARAVAL.Subindex = 16#00; FHPP+_I_Byte01.Subindex = 16#00; FHPP+_I_Byte02.Subindex = 16#00; FHPP+_I_Byte03.Subindex = 16#00; FHPP+_I_Byte04.Subindex = 16#00; FHPP+_I_Byte05.Subindex = 16#00; FHPP+_I_Byte06.Subindex = 16#00; FHPP+_I_Byte07.Subindex = 16#00; FHPP+_I_Byte08.Subindex = 16#00; FHPP+_I_Byte09.Subindex = 16#00; FHPP+_I_Byte10.Subindex = 16#00; FHPP+_I_Byte11.Subindex = 16#00; FHPP+_I_Byte12.Subindex = 16#00; FHPP+_I_Byte13.Subindex = 16#00; FHPP+_I_Byte14.Subindex = 16#00; FHPP+_I_Byte15.Subindex = 16#00; FHPP+_I_Byte16.Subindex = 16#00; SDO List.Disable TIME.Index = 16#1012; SDO List.Disable TIME.Subindex = 16#00; SDO List.Disable TIME.Value = 16#00000100; SDO List.Disable TIME.Size = 32; SDO List.Disable TIME.AbortIfError = FALSE; SDO List.Disable TIME.JumpToLine = FALSE; SDO List.Disable TIME.Line = 0; SDO List.Set Guardtime.Index = 16#100C; SDO List.Set Guardtime.Subindex = 16#00; SDO List.Set Guardtime.Value = 16#00000000; SDO List.Set Guardtime.Size = 16; SDO List.Set Guardtime.AbortIfError = FALSE; SDO List.Set Guardtime.JumpToLine = FALSE; SDO List.Set Guardtime.Line = 0;
              SDO List.Set Lifetime.Index = 16#100D; SDO List.Set Lifetime.Subindex = 16#00; SDO List.Set Lifetime.Value = 16#00000000; SDO List.Set Lifetime.Size = 8; SDO List.Set Lifetime.AbortIfError = FALSE; SDO List.Set Lifetime.JumpToLine = FALSE; SDO List.Set Lifetime.Line = 0; SDO List.Disable Emcy CobID.Index = 16#1014; SDO List.Disable Emcy CobID.Subindex = 16#00; SDO List.Disable Emcy CobID.Value = 16#80000081; SDO List.Disable Emcy CobID.Size = 32; SDO List.Disable Emcy CobID.AbortIfError = FALSE; SDO List.Disable Emcy CobID.JumpToLine = FALSE; SDO List.Disable Emcy CobID.Line = 0; SDO List.Set Emcy CobID.Index = 16#1014; SDO List.Set Emcy CobID.Subindex = 16#00; SDO List.Set Emcy CobID.Value = 16#00000081; SDO List.Set Emcy CobID.Size = 32; SDO List.Set Emcy CobID.AbortIfError = FALSE; SDO List.Set Emcy CobID.JumpToLine = FALSE; SDO List.Set Emcy CobID.Line = 0; SDO List.Set Heartbeat Consumer.Index = 16#1016; SDO List.Set Heartbeat Consumer.Subindex = 16#01; SDO List.Set Heartbeat Consumer.Value = 0; SDO List.Set Heartbeat Consumer.Size = 32; SDO List.Set Heartbeat Consumer.AbortIfError = FALSE; SDO List.Set Heartbeat Consumer.JumpToLine = FALSE; SDO List.Set Heartbeat Consumer.Line = 0; SDO List.Set Heartbeat Producer.Index = 16#1017; SDO List.Set Heartbeat Producer.Subindex = 16#00; SDO List.Set Heartbeat Producer.Value = 16#00000000; SDO List.Set Heartbeat Producer.Size = 16; SDO List.Set Heartbeat Producer.AbortIfError = FALSE; SDO List.Set Heartbeat Producer.JumpToLine = FALSE; SDO List.Set Heartbeat Producer.Line = 0; SDO List.Disable PDO.Index = 16#1400; SDO List.Disable PDO.Subindex = 16#01; SDO List.Disable PDO.Value = 16#80000201; SDO List.Disable PDO.Size = 32; SDO List.Disable PDO.AbortIfError = FALSE;
              SDO List.Disable PDO.JumpToLine = FALSE; SDO List.Disable PDO.Line = 0; SDO List.Set transmission type.Index = 16#1400; SDO List.Set transmission type.Subindex = 16#02; SDO List.Set transmission type.Value = 16#FF; SDO List.Set transmission type.Size = 8; SDO List.Set transmission type.AbortIfError = FALSE; SDO List.Set transmission type.JumpToLine = FALSE; SDO List.Set transmission type.Line = 0; SDO List.Set and enable COB-ID.Index = 16#1400; SDO List.Set and enable COB-ID.Subindex = 16#01; SDO List.Set and enable COB-ID.Value = 16#00000201; SDO List.Set and enable COB-ID.Size = 32; SDO List.Set and enable COB-ID.AbortIfError = FALSE; SDO List.Set and enable COB-ID.JumpToLine = FALSE; SDO List.Set and enable COB-ID.Line = 0; SDO List.Disable PDO.Index = 16#1401; SDO List.Disable PDO.Subindex = 16#01; SDO List.Disable PDO.Value = 16#80000301; SDO List.Disable PDO.Size = 32; SDO List.Disable PDO.AbortIfError = FALSE; SDO List.Disable PDO.JumpToLine = FALSE; SDO List.Disable PDO.Line = 0; SDO List.Set transmission type.Index = 16#1401; SDO List.Set transmission type.Subindex = 16#02; SDO List.Set transmission type.Value = 16#FF; SDO List.Set transmission type.Size = 8; SDO List.Set transmission type.AbortIfError = FALSE; SDO List.Set transmission type.JumpToLine = FALSE; SDO List.Set transmission type.Line = 0; SDO List.Set and enable COB-ID.Index = 16#1401; SDO List.Set and enable COB-ID.Subindex = 16#01; SDO List.Set and enable COB-ID.Value = 16#00000301; SDO List.Set and enable COB-ID.Size = 32; SDO List.Set and enable COB-ID.AbortIfError = FALSE; SDO List.Set and enable COB-ID.JumpToLine = FALSE; SDO List.Set and enable COB-ID.Line = 0; SDO List.Disable PDO.Index = 16#1402; SDO List.Disable PDO.Subindex = 16#01; SDO List.Disable PDO.Value = 16#80000401;
              SDO List.Disable PDO.Size = 32; SDO List.Disable PDO.AbortIfError = FALSE; SDO List.Disable PDO.JumpToLine = FALSE; SDO List.Disable PDO.Line = 0; SDO List.Set transmission type.Index = 16#1402; SDO List.Set transmission type.Subindex = 16#02; SDO List.Set transmission type.Value = 16#FF; SDO List.Set transmission type.Size = 8; SDO List.Set transmission type.AbortIfError = FALSE; SDO List.Set transmission type.JumpToLine = FALSE; SDO List.Set transmission type.Line = 0; SDO List.Clear pdo mapping.Index = 16#1602; SDO List.Clear pdo mapping.Subindex = 16#00; SDO List.Clear pdo mapping.Value = 16#0; SDO List.Clear pdo mapping.Size = 8; SDO List.Clear pdo mapping.AbortIfError = FALSE; SDO List.Clear pdo mapping.JumpToLine = FALSE; SDO List.Clear pdo mapping.Line = 0; SDO List.Set Mapping.Index = 16#1602; SDO List.Set Mapping.Subindex = 16#01; SDO List.Set Mapping.Value = 16#31010008; SDO List.Set Mapping.Size = 32; SDO List.Set Mapping.AbortIfError = FALSE; SDO List.Set Mapping.JumpToLine = FALSE; SDO List.Set Mapping.Line = 0; SDO List.Set Mapping.Index = 16#1602; SDO List.Set Mapping.Subindex = 16#02; SDO List.Set Mapping.Value = 16#31020008; SDO List.Set Mapping.Size = 32; SDO List.Set Mapping.AbortIfError = FALSE; SDO List.Set Mapping.JumpToLine = FALSE; SDO List.Set Mapping.Line = 0; SDO List.Set Mapping.Index = 16#1602; SDO List.Set Mapping.Subindex = 16#03; SDO List.Set Mapping.Value = 16#31030008; SDO List.Set Mapping.Size = 32; SDO List.Set Mapping.AbortIfError = FALSE; SDO List.Set Mapping.JumpToLine = FALSE; SDO List.Set Mapping.Line = 0; SDO List.Set Mapping.Index = 16#1602;
              SDO List.Set Mapping.Subindex = 16#04; SDO List.Set Mapping.Value = 16#31040008; SDO List.Set Mapping.Size = 32; SDO List.Set Mapping.AbortIfError = FALSE; SDO List.Set Mapping.JumpToLine = FALSE; SDO List.Set Mapping.Line = 0; SDO List.Set Mapping.Index = 16#1602; SDO List.Set Mapping.Subindex = 16#05; SDO List.Set Mapping.Value = 16#31050008; SDO List.Set Mapping.Size = 32; SDO List.Set Mapping.AbortIfError = FALSE; SDO List.Set Mapping.JumpToLine = FALSE; SDO List.Set Mapping.Line = 0; SDO List.Set Mapping.Index = 16#1602; SDO List.Set Mapping.Subindex = 16#06; SDO List.Set Mapping.Value = 16#31060008; SDO List.Set Mapping.Size = 32; SDO List.Set Mapping.AbortIfError = FALSE; SDO List.Set Mapping.JumpToLine = FALSE; SDO List.Set Mapping.Line = 0; SDO List.Set Mapping.Index = 16#1602; SDO List.Set Mapping.Subindex = 16#07; SDO List.Set Mapping.Value = 16#31070008; SDO List.Set Mapping.Size = 32; SDO List.Set Mapping.AbortIfError = FALSE; SDO List.Set Mapping.JumpToLine = FALSE; SDO List.Set Mapping.Line = 0; SDO List.Set Mapping.Index = 16#1602; SDO List.Set Mapping.Subindex = 16#08; SDO List.Set Mapping.Value = 16#31080008; SDO List.Set Mapping.Size = 32; SDO List.Set Mapping.AbortIfError = FALSE; SDO List.Set Mapping.JumpToLine = FALSE; SDO List.Set Mapping.Line = 0; SDO List.Set number of mappings.Index = 16#1602; SDO List.Set number of mappings.Subindex = 16#00; SDO List.Set number of mappings.Value = 16#08; SDO List.Set number of mappings.Size = 8; SDO List.Set number of mappings.AbortIfError = FALSE; SDO List.Set number of mappings.JumpToLine = FALSE;
              SDO List.Set number of mappings.Line = 0; SDO List.Set and enable COB-ID.Index = 16#1402; SDO List.Set and enable COB-ID.Subindex = 16#01; SDO List.Set and enable COB-ID.Value = 16#00000401; SDO List.Set and enable COB-ID.Size = 32; SDO List.Set and enable COB-ID.AbortIfError = FALSE; SDO List.Set and enable COB-ID.JumpToLine = FALSE; SDO List.Set and enable COB-ID.Line = 0; SDO List.Disable PDO.Index = 16#1403; SDO List.Disable PDO.Subindex = 16#01; SDO List.Disable PDO.Value = 16#80000501; SDO List.Disable PDO.Size = 32; SDO List.Disable PDO.AbortIfError = FALSE; SDO List.Disable PDO.JumpToLine = FALSE; SDO List.Disable PDO.Line = 0; SDO List.Set transmission type.Index = 16#1403; SDO List.Set transmission type.Subindex = 16#02; SDO List.Set transmission type.Value = 16#FF; SDO List.Set transmission type.Size = 8; SDO List.Set transmission type.AbortIfError = FALSE; SDO List.Set transmission type.JumpToLine = FALSE; SDO List.Set transmission type.Line = 0; SDO List.Clear pdo mapping.Index = 16#1603; SDO List.Clear pdo mapping.Subindex = 16#00; SDO List.Clear pdo mapping.Value = 16#0; SDO List.Clear pdo mapping.Size = 8; SDO List.Clear pdo mapping.AbortIfError = FALSE; SDO List.Clear pdo mapping.JumpToLine = FALSE; SDO List.Clear pdo mapping.Line = 0; SDO List.Set Mapping.Index = 16#1603; SDO List.Set Mapping.Subindex = 16#01; SDO List.Set Mapping.Value = 16#31090008; SDO List.Set Mapping.Size = 32; SDO List.Set Mapping.AbortIfError = FALSE; SDO List.Set Mapping.JumpToLine = FALSE; SDO List.Set Mapping.Line = 0; SDO List.Set Mapping.Index = 16#1603; SDO List.Set Mapping.Subindex = 16#02; SDO List.Set Mapping.Value = 16#31100008; SDO List.Set Mapping.Size = 32;
              SDO List.Set Mapping.AbortIfError = FALSE; SDO List.Set Mapping.JumpToLine = FALSE; SDO List.Set Mapping.Line = 0; SDO List.Set Mapping.Index = 16#1603; SDO List.Set Mapping.Subindex = 16#03; SDO List.Set Mapping.Value = 16#31110008; SDO List.Set Mapping.Size = 32; SDO List.Set Mapping.AbortIfError = FALSE; SDO List.Set Mapping.JumpToLine = FALSE; SDO List.Set Mapping.Line = 0; SDO List.Set Mapping.Index = 16#1603; SDO List.Set Mapping.Subindex = 16#04; SDO List.Set Mapping.Value = 16#31120008; SDO List.Set Mapping.Size = 32; SDO List.Set Mapping.AbortIfError = FALSE; SDO List.Set Mapping.JumpToLine = FALSE; SDO List.Set Mapping.Line = 0; SDO List.Set Mapping.Index = 16#1603; SDO List.Set Mapping.Subindex = 16#05; SDO List.Set Mapping.Value = 16#31130008; SDO List.Set Mapping.Size = 32; SDO List.Set Mapping.AbortIfError = FALSE; SDO List.Set Mapping.JumpToLine = FALSE; SDO List.Set Mapping.Line = 0; SDO List.Set Mapping.Index = 16#1603; SDO List.Set Mapping.Subindex = 16#06; SDO List.Set Mapping.Value = 16#31140008; SDO List.Set Mapping.Size = 32; SDO List.Set Mapping.AbortIfError = FALSE; SDO List.Set Mapping.JumpToLine = FALSE; SDO List.Set Mapping.Line = 0; SDO List.Set Mapping.Index = 16#1603; SDO List.Set Mapping.Subindex = 16#07; SDO List.Set Mapping.Value = 16#31150008; SDO List.Set Mapping.Size = 32; SDO List.Set Mapping.AbortIfError = FALSE; SDO List.Set Mapping.JumpToLine = FALSE; SDO List.Set Mapping.Line = 0; SDO List.Set Mapping.Index = 16#1603; SDO List.Set Mapping.Subindex = 16#08;
              SDO List.Set Mapping.Value = 16#31160008; SDO List.Set Mapping.Size = 32; SDO List.Set Mapping.AbortIfError = FALSE; SDO List.Set Mapping.JumpToLine = FALSE; SDO List.Set Mapping.Line = 0; SDO List.Set number of mappings.Index = 16#1603; SDO List.Set number of mappings.Subindex = 16#00; SDO List.Set number of mappings.Value = 16#08; SDO List.Set number of mappings.Size = 8; SDO List.Set number of mappings.AbortIfError = FALSE; SDO List.Set number of mappings.JumpToLine = FALSE; SDO List.Set number of mappings.Line = 0; SDO List.Set and enable COB-ID.Index = 16#1403; SDO List.Set and enable COB-ID.Subindex = 16#01; SDO List.Set and enable COB-ID.Value = 16#00000501; SDO List.Set and enable COB-ID.Size = 32; SDO List.Set and enable COB-ID.AbortIfError = FALSE; SDO List.Set and enable COB-ID.JumpToLine = FALSE; SDO List.Set and enable COB-ID.Line = 0; SDO List.Disable PDO.Index = 16#1800; SDO List.Disable PDO.Subindex = 16#01; SDO List.Disable PDO.Value = 16#80000181; SDO List.Disable PDO.Size = 32; SDO List.Disable PDO.AbortIfError = FALSE; SDO List.Disable PDO.JumpToLine = FALSE; SDO List.Disable PDO.Line = 0; SDO List.Set transmission type.Index = 16#1800; SDO List.Set transmission type.Subindex = 16#02; SDO List.Set transmission type.Value = 16#FF; SDO List.Set transmission type.Size = 8; SDO List.Set transmission type.AbortIfError = FALSE; SDO List.Set transmission type.JumpToLine = FALSE; SDO List.Set transmission type.Line = 0; SDO List.Set inhibit time.Index = 16#1800; SDO List.Set inhibit time.Subindex = 16#03; SDO List.Set inhibit time.Value = 16#0000; SDO List.Set inhibit time.Size = 16; SDO List.Set inhibit time.AbortIfError = FALSE; SDO List.Set inhibit time.JumpToLine = FALSE; SDO List.Set inhibit time.Line = 0;
              SDO List.Set and enable COB-ID.Index = 16#1800; SDO List.Set and enable COB-ID.Subindex = 16#01; SDO List.Set and enable COB-ID.Value = 16#00000181; SDO List.Set and enable COB-ID.Size = 32; SDO List.Set and enable COB-ID.AbortIfError = FALSE; SDO List.Set and enable COB-ID.JumpToLine = FALSE; SDO List.Set and enable COB-ID.Line = 0; SDO List.Disable PDO.Index = 16#1801; SDO List.Disable PDO.Subindex = 16#01; SDO List.Disable PDO.Value = 16#80000281; SDO List.Disable PDO.Size = 32; SDO List.Disable PDO.AbortIfError = FALSE; SDO List.Disable PDO.JumpToLine = FALSE; SDO List.Disable PDO.Line = 0; SDO List.Set transmission type.Index = 16#1801; SDO List.Set transmission type.Subindex = 16#02; SDO List.Set transmission type.Value = 16#FF; SDO List.Set transmission type.Size = 8; SDO List.Set transmission type.AbortIfError = FALSE; SDO List.Set transmission type.JumpToLine = FALSE; SDO List.Set transmission type.Line = 0; SDO List.Set inhibit time.Index = 16#1801; SDO List.Set inhibit time.Subindex = 16#03; SDO List.Set inhibit time.Value = 16#0000; SDO List.Set inhibit time.Size = 16; SDO List.Set inhibit time.AbortIfError = FALSE; SDO List.Set inhibit time.JumpToLine = FALSE; SDO List.Set inhibit time.Line = 0; SDO List.Set and enable COB-ID.Index = 16#1801; SDO List.Set and enable COB-ID.Subindex = 16#01; SDO List.Set and enable COB-ID.Value = 16#00000281; SDO List.Set and enable COB-ID.Size = 32; SDO List.Set and enable COB-ID.AbortIfError = FALSE; SDO List.Set and enable COB-ID.JumpToLine = FALSE; SDO List.Set and enable COB-ID.Line = 0; SDO List.Disable PDO.Index = 16#1802; SDO List.Disable PDO.Subindex = 16#01; SDO List.Disable PDO.Value = 16#80000381; SDO List.Disable PDO.Size = 32; SDO List.Disable PDO.AbortIfError = FALSE;
              SDO List.Disable PDO.JumpToLine = FALSE; SDO List.Disable PDO.Line = 0; SDO List.Set transmission type.Index = 16#1802; SDO List.Set transmission type.Subindex = 16#02; SDO List.Set transmission type.Value = 16#FF; SDO List.Set transmission type.Size = 8; SDO List.Set transmission type.AbortIfError = FALSE; SDO List.Set transmission type.JumpToLine = FALSE; SDO List.Set transmission type.Line = 0; SDO List.Set inhibit time.Index = 16#1802; SDO List.Set inhibit time.Subindex = 16#03; SDO List.Set inhibit time.Value = 16#0000; SDO List.Set inhibit time.Size = 16; SDO List.Set inhibit time.AbortIfError = FALSE; SDO List.Set inhibit time.JumpToLine = FALSE; SDO List.Set inhibit time.Line = 0; SDO List.Clear pdo mapping.Index = 16#1A02; SDO List.Clear pdo mapping.Subindex = 16#00; SDO List.Clear pdo mapping.Value = 16#0; SDO List.Clear pdo mapping.Size = 8; SDO List.Clear pdo mapping.AbortIfError = FALSE; SDO List.Clear pdo mapping.JumpToLine = FALSE; SDO List.Clear pdo mapping.Line = 0; SDO List.Set Mapping.Index = 16#1A02; SDO List.Set Mapping.Subindex = 16#01; SDO List.Set Mapping.Value = 16#32010008; SDO List.Set Mapping.Size = 32; SDO List.Set Mapping.AbortIfError = FALSE; SDO List.Set Mapping.JumpToLine = FALSE; SDO List.Set Mapping.Line = 0; SDO List.Set Mapping.Index = 16#1A02; SDO List.Set Mapping.Subindex = 16#02; SDO List.Set Mapping.Value = 16#32020008; SDO List.Set Mapping.Size = 32; SDO List.Set Mapping.AbortIfError = FALSE; SDO List.Set Mapping.JumpToLine = FALSE; SDO List.Set Mapping.Line = 0; SDO List.Set Mapping.Index = 16#1A02; SDO List.Set Mapping.Subindex = 16#03; SDO List.Set Mapping.Value = 16#32030008;
              SDO List.Set Mapping.Size = 32; SDO List.Set Mapping.AbortIfError = FALSE; SDO List.Set Mapping.JumpToLine = FALSE; SDO List.Set Mapping.Line = 0; SDO List.Set Mapping.Index = 16#1A02; SDO List.Set Mapping.Subindex = 16#04; SDO List.Set Mapping.Value = 16#32040008; SDO List.Set Mapping.Size = 32; SDO List.Set Mapping.AbortIfError = FALSE; SDO List.Set Mapping.JumpToLine = FALSE; SDO List.Set Mapping.Line = 0; SDO List.Set Mapping.Index = 16#1A02; SDO List.Set Mapping.Subindex = 16#05; SDO List.Set Mapping.Value = 16#32050008; SDO List.Set Mapping.Size = 32; SDO List.Set Mapping.AbortIfError = FALSE; SDO List.Set Mapping.JumpToLine = FALSE; SDO List.Set Mapping.Line = 0; SDO List.Set Mapping.Index = 16#1A02; SDO List.Set Mapping.Subindex = 16#06; SDO List.Set Mapping.Value = 16#32060008; SDO List.Set Mapping.Size = 32; SDO List.Set Mapping.AbortIfError = FALSE; SDO List.Set Mapping.JumpToLine = FALSE; SDO List.Set Mapping.Line = 0; SDO List.Set Mapping.Index = 16#1A02; SDO List.Set Mapping.Subindex = 16#07; SDO List.Set Mapping.Value = 16#32070008; SDO List.Set Mapping.Size = 32; SDO List.Set Mapping.AbortIfError = FALSE; SDO List.Set Mapping.JumpToLine = FALSE; SDO List.Set Mapping.Line = 0; SDO List.Set Mapping.Index = 16#1A02; SDO List.Set Mapping.Subindex = 16#08; SDO List.Set Mapping.Value = 16#32080008; SDO List.Set Mapping.Size = 32; SDO List.Set Mapping.AbortIfError = FALSE; SDO List.Set Mapping.JumpToLine = FALSE; SDO List.Set Mapping.Line = 0; SDO List.Set number of mappings.Index = 16#1A02;
              SDO List.Set number of mappings.Subindex = 16#00; SDO List.Set number of mappings.Value = 16#08; SDO List.Set number of mappings.Size = 8; SDO List.Set number of mappings.AbortIfError = FALSE; SDO List.Set number of mappings.JumpToLine = FALSE; SDO List.Set number of mappings.Line = 0; SDO List.Set and enable COB-ID.Index = 16#1802; SDO List.Set and enable COB-ID.Subindex = 16#01; SDO List.Set and enable COB-ID.Value = 16#00000381; SDO List.Set and enable COB-ID.Size = 32; SDO List.Set and enable COB-ID.AbortIfError = FALSE; SDO List.Set and enable COB-ID.JumpToLine = FALSE; SDO List.Set and enable COB-ID.Line = 0; SDO List.Disable PDO.Index = 16#1803; SDO List.Disable PDO.Subindex = 16#01; SDO List.Disable PDO.Value = 16#80000481; SDO List.Disable PDO.Size = 32; SDO List.Disable PDO.AbortIfError = FALSE; SDO List.Disable PDO.JumpToLine = FALSE; SDO List.Disable PDO.Line = 0; SDO List.Set transmission type.Index = 16#1803; SDO List.Set transmission type.Subindex = 16#02; SDO List.Set transmission type.Value = 16#FF; SDO List.Set transmission type.Size = 8; SDO List.Set transmission type.AbortIfError = FALSE; SDO List.Set transmission type.JumpToLine = FALSE; SDO List.Set transmission type.Line = 0; SDO List.Set inhibit time.Index = 16#1803; SDO List.Set inhibit time.Subindex = 16#03; SDO List.Set inhibit time.Value = 16#0000; SDO List.Set inhibit time.Size = 16; SDO List.Set inhibit time.AbortIfError = FALSE; SDO List.Set inhibit time.JumpToLine = FALSE; SDO List.Set inhibit time.Line = 0; SDO List.Clear pdo mapping.Index = 16#1A03; SDO List.Clear pdo mapping.Subindex = 16#00; SDO List.Clear pdo mapping.Value = 16#0; SDO List.Clear pdo mapping.Size = 8; SDO List.Clear pdo mapping.AbortIfError = FALSE; SDO List.Clear pdo mapping.JumpToLine = FALSE;
              SDO List.Clear pdo mapping.Line = 0; SDO List.Set Mapping.Index = 16#1A03; SDO List.Set Mapping.Subindex = 16#01; SDO List.Set Mapping.Value = 16#32090008; SDO List.Set Mapping.Size = 32; SDO List.Set Mapping.AbortIfError = FALSE; SDO List.Set Mapping.JumpToLine = FALSE; SDO List.Set Mapping.Line = 0; SDO List.Set Mapping.Index = 16#1A03; SDO List.Set Mapping.Subindex = 16#02; SDO List.Set Mapping.Value = 16#32100008; SDO List.Set Mapping.Size = 32; SDO List.Set Mapping.AbortIfError = FALSE; SDO List.Set Mapping.JumpToLine = FALSE; SDO List.Set Mapping.Line = 0; SDO List.Set Mapping.Index = 16#1A03; SDO List.Set Mapping.Subindex = 16#03; SDO List.Set Mapping.Value = 16#32110008; SDO List.Set Mapping.Size = 32; SDO List.Set Mapping.AbortIfError = FALSE; SDO List.Set Mapping.JumpToLine = FALSE; SDO List.Set Mapping.Line = 0; SDO List.Set Mapping.Index = 16#1A03; SDO List.Set Mapping.Subindex = 16#04; SDO List.Set Mapping.Value = 16#32120008; SDO List.Set Mapping.Size = 32; SDO List.Set Mapping.AbortIfError = FALSE; SDO List.Set Mapping.JumpToLine = FALSE; SDO List.Set Mapping.Line = 0; SDO List.Set Mapping.Index = 16#1A03; SDO List.Set Mapping.Subindex = 16#05; SDO List.Set Mapping.Value = 16#32130008; SDO List.Set Mapping.Size = 32; SDO List.Set Mapping.AbortIfError = FALSE; SDO List.Set Mapping.JumpToLine = FALSE; SDO List.Set Mapping.Line = 0; SDO List.Set Mapping.Index = 16#1A03; SDO List.Set Mapping.Subindex = 16#06; SDO List.Set Mapping.Value = 16#32140008; SDO List.Set Mapping.Size = 32;
              SDO List.Set Mapping.AbortIfError = FALSE; SDO List.Set Mapping.JumpToLine = FALSE; SDO List.Set Mapping.Line = 0; SDO List.Set Mapping.Index = 16#1A03; SDO List.Set Mapping.Subindex = 16#07; SDO List.Set Mapping.Value = 16#32150008; SDO List.Set Mapping.Size = 32; SDO List.Set Mapping.AbortIfError = FALSE; SDO List.Set Mapping.JumpToLine = FALSE; SDO List.Set Mapping.Line = 0; SDO List.Set Mapping.Index = 16#1A03; SDO List.Set Mapping.Subindex = 16#08; SDO List.Set Mapping.Value = 16#32160008; SDO List.Set Mapping.Size = 32; SDO List.Set Mapping.AbortIfError = FALSE; SDO List.Set Mapping.JumpToLine = FALSE; SDO List.Set Mapping.Line = 0; SDO List.Set number of mappings.Index = 16#1A03; SDO List.Set number of mappings.Subindex = 16#00; SDO List.Set number of mappings.Value = 16#08; SDO List.Set number of mappings.Size = 8; SDO List.Set number of mappings.AbortIfError = FALSE; SDO List.Set number of mappings.JumpToLine = FALSE; SDO List.Set number of mappings.Line = 0; SDO List.Set and enable COB-ID.Index = 16#1803; SDO List.Set and enable COB-ID.Subindex = 16#01; SDO List.Set and enable COB-ID.Value = 16#00000481; SDO List.Set and enable COB-ID.Size = 32; SDO List.Set and enable COB-ID.AbortIfError = FALSE; SDO List.Set and enable COB-ID.JumpToLine = FALSE; SDO List.Set and enable COB-ID.Line = 0; ConfigVersion = 50659584
            unmapped channels: CCON, CPOS, REC_NR/CDIR, RES/DEM_VAL1/PARA1, RES/DEM_VAL2/PARA2, RES, SUBINDEX, REQCODE_PNU, PARAVAL, FHPP+_O_Byte01, FHPP+_O_Byte02, FHPP+_O_Byte03, FHPP+_O_Byte04, FHPP+_O_Byte05, FHPP+_O_Byte06, FHPP+_O_Byte07, FHPP+_O_Byte08, FHPP+_O_Byte09, FHPP+_O_Byte10, FHPP+_O_Byte11, FHPP+_O_Byte12, FHPP+_O_Byte13, FHPP+_O_Byte14, FHPP+_O_Byte15, FHPP+_O_Byte16, SCON, SPOS, REC_NR/SDIR, RSB/ACT_VAL1, ACT_POS/ACT_VAL2, RES, SUBINDEX, RESPCODE_PNU, PARAVAL, FHPP+_I_Byte01, FHPP+_I_Byte02, FHPP+_I_Byte03, FHPP+_I_Byte04, FHPP+_I_Byte05, FHPP+_I_Byte06,
              FHPP+_I_Byte07, FHPP+_I_Byte08, FHPP+_I_Byte09, FHPP+_I_Byte10, FHPP+_I_Byte11, FHPP+_I_Byte12, FHPP+_I_Byte13, FHPP+_I_Byte14, FHPP+_I_Byte15, FHPP+_I_Byte16
        U2 : CMMP-AS-C5-3A-M0 (FHPP), Festo AG & Co. KG, order no. 1622902, version 0.262146.CMMP_AS_C5_3A_M0_FHPP.2.8
            settings: General Options.Reset Node = FALSE; NODEIDSAVED = 2; SDO Timeout = 1000000; PDO_Autoconfig = FALSE; EXPERTSETTINGS = TRUE; Emergency-General Parameters.Emergency COBID = 16#00000082; PDO 16#1400.COBID = 16#00000202; PDO 16#1401.COBID = 16#00000302; PDO 16#1402.COBID = 16#00000402; PDO 16#1403.COBID = 16#00000502; PDO 16#1800.COBID = 16#00000182; PDO 16#1800.Event Timer = 0; PDO 16#1801.COBID = 16#00000282; PDO 16#1801.Event Timer = 0; PDO 16#1802.COBID = 16#00000382; PDO 16#1802.Event Timer = 0; PDO 16#1803.COBID = 16#00000482; PDO 16#1803.Event Timer = 0; CCON.Subindex = 16#00; CPOS.Subindex = 16#00; REC_NR/CDIR.Subindex = 16#00; RES/DEM_VAL1/PARA1.Subindex = 16#00; RES/DEM_VAL2/PARA2.Subindex = 16#00; RES.Subindex = 16#00; SUBINDEX.Subindex = 16#00; REQCODE_PNU.Subindex = 16#00; PARAVAL.Subindex = 16#00; FHPP+_O_Byte01.Subindex = 16#00; FHPP+_O_Byte02.Subindex = 16#00; FHPP+_O_Byte03.Subindex = 16#00; FHPP+_O_Byte04.Subindex = 16#00; FHPP+_O_Byte05.Subindex = 16#00; FHPP+_O_Byte06.Subindex = 16#00; FHPP+_O_Byte07.Subindex = 16#00; FHPP+_O_Byte08.Subindex = 16#00; FHPP+_O_Byte09.Subindex = 16#00; FHPP+_O_Byte10.Subindex = 16#00; FHPP+_O_Byte11.Subindex = 16#00; FHPP+_O_Byte12.Subindex = 16#00; FHPP+_O_Byte13.Subindex = 16#00;
              FHPP+_O_Byte14.Subindex = 16#00; FHPP+_O_Byte15.Subindex = 16#00; FHPP+_O_Byte16.Subindex = 16#00; SCON.Subindex = 16#00; SPOS.Subindex = 16#00; REC_NR/SDIR.Subindex = 16#00; RSB/ACT_VAL1.Subindex = 16#00; ACT_POS/ACT_VAL2.Subindex = 16#00; RES.Subindex = 16#00; SUBINDEX.Subindex = 16#00; RESPCODE_PNU.Subindex = 16#00; PARAVAL.Subindex = 16#00; FHPP+_I_Byte01.Subindex = 16#00; FHPP+_I_Byte02.Subindex = 16#00; FHPP+_I_Byte03.Subindex = 16#00; FHPP+_I_Byte04.Subindex = 16#00; FHPP+_I_Byte05.Subindex = 16#00; FHPP+_I_Byte06.Subindex = 16#00; FHPP+_I_Byte07.Subindex = 16#00; FHPP+_I_Byte08.Subindex = 16#00; FHPP+_I_Byte09.Subindex = 16#00; FHPP+_I_Byte10.Subindex = 16#00; FHPP+_I_Byte11.Subindex = 16#00; FHPP+_I_Byte12.Subindex = 16#00; FHPP+_I_Byte13.Subindex = 16#00; FHPP+_I_Byte14.Subindex = 16#00; FHPP+_I_Byte15.Subindex = 16#00; FHPP+_I_Byte16.Subindex = 16#00; SDO List.Disable TIME.Index = 16#1012; SDO List.Disable TIME.Subindex = 16#00; SDO List.Disable TIME.Value = 16#00000100; SDO List.Disable TIME.Size = 32; SDO List.Disable TIME.AbortIfError = FALSE; SDO List.Disable TIME.JumpToLine = FALSE; SDO List.Disable TIME.Line = 0; SDO List.Set Guardtime.Index = 16#100C; SDO List.Set Guardtime.Subindex = 16#00; SDO List.Set Guardtime.Value = 16#00000000; SDO List.Set Guardtime.Size = 16; SDO List.Set Guardtime.AbortIfError = FALSE;
              SDO List.Set Guardtime.JumpToLine = FALSE; SDO List.Set Guardtime.Line = 0; SDO List.Set Lifetime.Index = 16#100D; SDO List.Set Lifetime.Subindex = 16#00; SDO List.Set Lifetime.Value = 16#00000000; SDO List.Set Lifetime.Size = 8; SDO List.Set Lifetime.AbortIfError = FALSE; SDO List.Set Lifetime.JumpToLine = FALSE; SDO List.Set Lifetime.Line = 0; SDO List.Disable Emcy CobID.Index = 16#1014; SDO List.Disable Emcy CobID.Subindex = 16#00; SDO List.Disable Emcy CobID.Value = 16#80000082; SDO List.Disable Emcy CobID.Size = 32; SDO List.Disable Emcy CobID.AbortIfError = FALSE; SDO List.Disable Emcy CobID.JumpToLine = FALSE; SDO List.Disable Emcy CobID.Line = 0; SDO List.Set Emcy CobID.Index = 16#1014; SDO List.Set Emcy CobID.Subindex = 16#00; SDO List.Set Emcy CobID.Value = 16#00000082; SDO List.Set Emcy CobID.Size = 32; SDO List.Set Emcy CobID.AbortIfError = FALSE; SDO List.Set Emcy CobID.JumpToLine = FALSE; SDO List.Set Emcy CobID.Line = 0; SDO List.Set Heartbeat Consumer.Index = 16#1016; SDO List.Set Heartbeat Consumer.Subindex = 16#01; SDO List.Set Heartbeat Consumer.Value = 0; SDO List.Set Heartbeat Consumer.Size = 32; SDO List.Set Heartbeat Consumer.AbortIfError = FALSE; SDO List.Set Heartbeat Consumer.JumpToLine = FALSE; SDO List.Set Heartbeat Consumer.Line = 0; SDO List.Set Heartbeat Producer.Index = 16#1017; SDO List.Set Heartbeat Producer.Subindex = 16#00; SDO List.Set Heartbeat Producer.Value = 16#00000000; SDO List.Set Heartbeat Producer.Size = 16; SDO List.Set Heartbeat Producer.AbortIfError = FALSE; SDO List.Set Heartbeat Producer.JumpToLine = FALSE; SDO List.Set Heartbeat Producer.Line = 0; SDO List.Disable PDO.Index = 16#1400; SDO List.Disable PDO.Subindex = 16#01; SDO List.Disable PDO.Value = 16#80000202;
              SDO List.Disable PDO.Size = 32; SDO List.Disable PDO.AbortIfError = FALSE; SDO List.Disable PDO.JumpToLine = FALSE; SDO List.Disable PDO.Line = 0; SDO List.Set transmission type.Index = 16#1400; SDO List.Set transmission type.Subindex = 16#02; SDO List.Set transmission type.Value = 16#FF; SDO List.Set transmission type.Size = 8; SDO List.Set transmission type.AbortIfError = FALSE; SDO List.Set transmission type.JumpToLine = FALSE; SDO List.Set transmission type.Line = 0; SDO List.Set and enable COB-ID.Index = 16#1400; SDO List.Set and enable COB-ID.Subindex = 16#01; SDO List.Set and enable COB-ID.Value = 16#00000202; SDO List.Set and enable COB-ID.Size = 32; SDO List.Set and enable COB-ID.AbortIfError = FALSE; SDO List.Set and enable COB-ID.JumpToLine = FALSE; SDO List.Set and enable COB-ID.Line = 0; SDO List.Disable PDO.Index = 16#1401; SDO List.Disable PDO.Subindex = 16#01; SDO List.Disable PDO.Value = 16#80000302; SDO List.Disable PDO.Size = 32; SDO List.Disable PDO.AbortIfError = FALSE; SDO List.Disable PDO.JumpToLine = FALSE; SDO List.Disable PDO.Line = 0; SDO List.Set transmission type.Index = 16#1401; SDO List.Set transmission type.Subindex = 16#02; SDO List.Set transmission type.Value = 16#FF; SDO List.Set transmission type.Size = 8; SDO List.Set transmission type.AbortIfError = FALSE; SDO List.Set transmission type.JumpToLine = FALSE; SDO List.Set transmission type.Line = 0; SDO List.Set and enable COB-ID.Index = 16#1401; SDO List.Set and enable COB-ID.Subindex = 16#01; SDO List.Set and enable COB-ID.Value = 16#00000302; SDO List.Set and enable COB-ID.Size = 32; SDO List.Set and enable COB-ID.AbortIfError = FALSE; SDO List.Set and enable COB-ID.JumpToLine = FALSE; SDO List.Set and enable COB-ID.Line = 0; SDO List.Disable PDO.Index = 16#1402;
              SDO List.Disable PDO.Subindex = 16#01; SDO List.Disable PDO.Value = 16#80000402; SDO List.Disable PDO.Size = 32; SDO List.Disable PDO.AbortIfError = FALSE; SDO List.Disable PDO.JumpToLine = FALSE; SDO List.Disable PDO.Line = 0; SDO List.Set transmission type.Index = 16#1402; SDO List.Set transmission type.Subindex = 16#02; SDO List.Set transmission type.Value = 16#FF; SDO List.Set transmission type.Size = 8; SDO List.Set transmission type.AbortIfError = FALSE; SDO List.Set transmission type.JumpToLine = FALSE; SDO List.Set transmission type.Line = 0; SDO List.Clear pdo mapping.Index = 16#1602; SDO List.Clear pdo mapping.Subindex = 16#00; SDO List.Clear pdo mapping.Value = 16#0; SDO List.Clear pdo mapping.Size = 8; SDO List.Clear pdo mapping.AbortIfError = FALSE; SDO List.Clear pdo mapping.JumpToLine = FALSE; SDO List.Clear pdo mapping.Line = 0; SDO List.Set Mapping.Index = 16#1602; SDO List.Set Mapping.Subindex = 16#01; SDO List.Set Mapping.Value = 16#31010008; SDO List.Set Mapping.Size = 32; SDO List.Set Mapping.AbortIfError = FALSE; SDO List.Set Mapping.JumpToLine = FALSE; SDO List.Set Mapping.Line = 0; SDO List.Set Mapping.Index = 16#1602; SDO List.Set Mapping.Subindex = 16#02; SDO List.Set Mapping.Value = 16#31020008; SDO List.Set Mapping.Size = 32; SDO List.Set Mapping.AbortIfError = FALSE; SDO List.Set Mapping.JumpToLine = FALSE; SDO List.Set Mapping.Line = 0; SDO List.Set Mapping.Index = 16#1602; SDO List.Set Mapping.Subindex = 16#03; SDO List.Set Mapping.Value = 16#31030008; SDO List.Set Mapping.Size = 32; SDO List.Set Mapping.AbortIfError = FALSE; SDO List.Set Mapping.JumpToLine = FALSE;
              SDO List.Set Mapping.Line = 0; SDO List.Set Mapping.Index = 16#1602; SDO List.Set Mapping.Subindex = 16#04; SDO List.Set Mapping.Value = 16#31040008; SDO List.Set Mapping.Size = 32; SDO List.Set Mapping.AbortIfError = FALSE; SDO List.Set Mapping.JumpToLine = FALSE; SDO List.Set Mapping.Line = 0; SDO List.Set Mapping.Index = 16#1602; SDO List.Set Mapping.Subindex = 16#05; SDO List.Set Mapping.Value = 16#31050008; SDO List.Set Mapping.Size = 32; SDO List.Set Mapping.AbortIfError = FALSE; SDO List.Set Mapping.JumpToLine = FALSE; SDO List.Set Mapping.Line = 0; SDO List.Set Mapping.Index = 16#1602; SDO List.Set Mapping.Subindex = 16#06; SDO List.Set Mapping.Value = 16#31060008; SDO List.Set Mapping.Size = 32; SDO List.Set Mapping.AbortIfError = FALSE; SDO List.Set Mapping.JumpToLine = FALSE; SDO List.Set Mapping.Line = 0; SDO List.Set Mapping.Index = 16#1602; SDO List.Set Mapping.Subindex = 16#07; SDO List.Set Mapping.Value = 16#31070008; SDO List.Set Mapping.Size = 32; SDO List.Set Mapping.AbortIfError = FALSE; SDO List.Set Mapping.JumpToLine = FALSE; SDO List.Set Mapping.Line = 0; SDO List.Set Mapping.Index = 16#1602; SDO List.Set Mapping.Subindex = 16#08; SDO List.Set Mapping.Value = 16#31080008; SDO List.Set Mapping.Size = 32; SDO List.Set Mapping.AbortIfError = FALSE; SDO List.Set Mapping.JumpToLine = FALSE; SDO List.Set Mapping.Line = 0; SDO List.Set number of mappings.Index = 16#1602; SDO List.Set number of mappings.Subindex = 16#00; SDO List.Set number of mappings.Value = 16#08; SDO List.Set number of mappings.Size = 8;
              SDO List.Set number of mappings.AbortIfError = FALSE; SDO List.Set number of mappings.JumpToLine = FALSE; SDO List.Set number of mappings.Line = 0; SDO List.Set and enable COB-ID.Index = 16#1402; SDO List.Set and enable COB-ID.Subindex = 16#01; SDO List.Set and enable COB-ID.Value = 16#00000402; SDO List.Set and enable COB-ID.Size = 32; SDO List.Set and enable COB-ID.AbortIfError = FALSE; SDO List.Set and enable COB-ID.JumpToLine = FALSE; SDO List.Set and enable COB-ID.Line = 0; SDO List.Disable PDO.Index = 16#1403; SDO List.Disable PDO.Subindex = 16#01; SDO List.Disable PDO.Value = 16#80000502; SDO List.Disable PDO.Size = 32; SDO List.Disable PDO.AbortIfError = FALSE; SDO List.Disable PDO.JumpToLine = FALSE; SDO List.Disable PDO.Line = 0; SDO List.Set transmission type.Index = 16#1403; SDO List.Set transmission type.Subindex = 16#02; SDO List.Set transmission type.Value = 16#FF; SDO List.Set transmission type.Size = 8; SDO List.Set transmission type.AbortIfError = FALSE; SDO List.Set transmission type.JumpToLine = FALSE; SDO List.Set transmission type.Line = 0; SDO List.Clear pdo mapping.Index = 16#1603; SDO List.Clear pdo mapping.Subindex = 16#00; SDO List.Clear pdo mapping.Value = 16#0; SDO List.Clear pdo mapping.Size = 8; SDO List.Clear pdo mapping.AbortIfError = FALSE; SDO List.Clear pdo mapping.JumpToLine = FALSE; SDO List.Clear pdo mapping.Line = 0; SDO List.Set Mapping.Index = 16#1603; SDO List.Set Mapping.Subindex = 16#01; SDO List.Set Mapping.Value = 16#31090008; SDO List.Set Mapping.Size = 32; SDO List.Set Mapping.AbortIfError = FALSE; SDO List.Set Mapping.JumpToLine = FALSE; SDO List.Set Mapping.Line = 0; SDO List.Set Mapping.Index = 16#1603; SDO List.Set Mapping.Subindex = 16#02;
              SDO List.Set Mapping.Value = 16#31100008; SDO List.Set Mapping.Size = 32; SDO List.Set Mapping.AbortIfError = FALSE; SDO List.Set Mapping.JumpToLine = FALSE; SDO List.Set Mapping.Line = 0; SDO List.Set Mapping.Index = 16#1603; SDO List.Set Mapping.Subindex = 16#03; SDO List.Set Mapping.Value = 16#31110008; SDO List.Set Mapping.Size = 32; SDO List.Set Mapping.AbortIfError = FALSE; SDO List.Set Mapping.JumpToLine = FALSE; SDO List.Set Mapping.Line = 0; SDO List.Set Mapping.Index = 16#1603; SDO List.Set Mapping.Subindex = 16#04; SDO List.Set Mapping.Value = 16#31120008; SDO List.Set Mapping.Size = 32; SDO List.Set Mapping.AbortIfError = FALSE; SDO List.Set Mapping.JumpToLine = FALSE; SDO List.Set Mapping.Line = 0; SDO List.Set Mapping.Index = 16#1603; SDO List.Set Mapping.Subindex = 16#05; SDO List.Set Mapping.Value = 16#31130008; SDO List.Set Mapping.Size = 32; SDO List.Set Mapping.AbortIfError = FALSE; SDO List.Set Mapping.JumpToLine = FALSE; SDO List.Set Mapping.Line = 0; SDO List.Set Mapping.Index = 16#1603; SDO List.Set Mapping.Subindex = 16#06; SDO List.Set Mapping.Value = 16#31140008; SDO List.Set Mapping.Size = 32; SDO List.Set Mapping.AbortIfError = FALSE; SDO List.Set Mapping.JumpToLine = FALSE; SDO List.Set Mapping.Line = 0; SDO List.Set Mapping.Index = 16#1603; SDO List.Set Mapping.Subindex = 16#07; SDO List.Set Mapping.Value = 16#31150008; SDO List.Set Mapping.Size = 32; SDO List.Set Mapping.AbortIfError = FALSE; SDO List.Set Mapping.JumpToLine = FALSE; SDO List.Set Mapping.Line = 0;
              SDO List.Set Mapping.Index = 16#1603; SDO List.Set Mapping.Subindex = 16#08; SDO List.Set Mapping.Value = 16#31160008; SDO List.Set Mapping.Size = 32; SDO List.Set Mapping.AbortIfError = FALSE; SDO List.Set Mapping.JumpToLine = FALSE; SDO List.Set Mapping.Line = 0; SDO List.Set number of mappings.Index = 16#1603; SDO List.Set number of mappings.Subindex = 16#00; SDO List.Set number of mappings.Value = 16#08; SDO List.Set number of mappings.Size = 8; SDO List.Set number of mappings.AbortIfError = FALSE; SDO List.Set number of mappings.JumpToLine = FALSE; SDO List.Set number of mappings.Line = 0; SDO List.Set and enable COB-ID.Index = 16#1403; SDO List.Set and enable COB-ID.Subindex = 16#01; SDO List.Set and enable COB-ID.Value = 16#00000502; SDO List.Set and enable COB-ID.Size = 32; SDO List.Set and enable COB-ID.AbortIfError = FALSE; SDO List.Set and enable COB-ID.JumpToLine = FALSE; SDO List.Set and enable COB-ID.Line = 0; SDO List.Disable PDO.Index = 16#1800; SDO List.Disable PDO.Subindex = 16#01; SDO List.Disable PDO.Value = 16#80000182; SDO List.Disable PDO.Size = 32; SDO List.Disable PDO.AbortIfError = FALSE; SDO List.Disable PDO.JumpToLine = FALSE; SDO List.Disable PDO.Line = 0; SDO List.Set transmission type.Index = 16#1800; SDO List.Set transmission type.Subindex = 16#02; SDO List.Set transmission type.Value = 16#FF; SDO List.Set transmission type.Size = 8; SDO List.Set transmission type.AbortIfError = FALSE; SDO List.Set transmission type.JumpToLine = FALSE; SDO List.Set transmission type.Line = 0; SDO List.Set inhibit time.Index = 16#1800; SDO List.Set inhibit time.Subindex = 16#03; SDO List.Set inhibit time.Value = 16#0000; SDO List.Set inhibit time.Size = 16; SDO List.Set inhibit time.AbortIfError = FALSE;
              SDO List.Set inhibit time.JumpToLine = FALSE; SDO List.Set inhibit time.Line = 0; SDO List.Set and enable COB-ID.Index = 16#1800; SDO List.Set and enable COB-ID.Subindex = 16#01; SDO List.Set and enable COB-ID.Value = 16#00000182; SDO List.Set and enable COB-ID.Size = 32; SDO List.Set and enable COB-ID.AbortIfError = FALSE; SDO List.Set and enable COB-ID.JumpToLine = FALSE; SDO List.Set and enable COB-ID.Line = 0; SDO List.Disable PDO.Index = 16#1801; SDO List.Disable PDO.Subindex = 16#01; SDO List.Disable PDO.Value = 16#80000282; SDO List.Disable PDO.Size = 32; SDO List.Disable PDO.AbortIfError = FALSE; SDO List.Disable PDO.JumpToLine = FALSE; SDO List.Disable PDO.Line = 0; SDO List.Set transmission type.Index = 16#1801; SDO List.Set transmission type.Subindex = 16#02; SDO List.Set transmission type.Value = 16#FF; SDO List.Set transmission type.Size = 8; SDO List.Set transmission type.AbortIfError = FALSE; SDO List.Set transmission type.JumpToLine = FALSE; SDO List.Set transmission type.Line = 0; SDO List.Set inhibit time.Index = 16#1801; SDO List.Set inhibit time.Subindex = 16#03; SDO List.Set inhibit time.Value = 16#0000; SDO List.Set inhibit time.Size = 16; SDO List.Set inhibit time.AbortIfError = FALSE; SDO List.Set inhibit time.JumpToLine = FALSE; SDO List.Set inhibit time.Line = 0; SDO List.Set and enable COB-ID.Index = 16#1801; SDO List.Set and enable COB-ID.Subindex = 16#01; SDO List.Set and enable COB-ID.Value = 16#00000282; SDO List.Set and enable COB-ID.Size = 32; SDO List.Set and enable COB-ID.AbortIfError = FALSE; SDO List.Set and enable COB-ID.JumpToLine = FALSE; SDO List.Set and enable COB-ID.Line = 0; SDO List.Disable PDO.Index = 16#1802; SDO List.Disable PDO.Subindex = 16#01; SDO List.Disable PDO.Value = 16#80000382;
              SDO List.Disable PDO.Size = 32; SDO List.Disable PDO.AbortIfError = FALSE; SDO List.Disable PDO.JumpToLine = FALSE; SDO List.Disable PDO.Line = 0; SDO List.Set transmission type.Index = 16#1802; SDO List.Set transmission type.Subindex = 16#02; SDO List.Set transmission type.Value = 16#FF; SDO List.Set transmission type.Size = 8; SDO List.Set transmission type.AbortIfError = FALSE; SDO List.Set transmission type.JumpToLine = FALSE; SDO List.Set transmission type.Line = 0; SDO List.Set inhibit time.Index = 16#1802; SDO List.Set inhibit time.Subindex = 16#03; SDO List.Set inhibit time.Value = 16#0000; SDO List.Set inhibit time.Size = 16; SDO List.Set inhibit time.AbortIfError = FALSE; SDO List.Set inhibit time.JumpToLine = FALSE; SDO List.Set inhibit time.Line = 0; SDO List.Clear pdo mapping.Index = 16#1A02; SDO List.Clear pdo mapping.Subindex = 16#00; SDO List.Clear pdo mapping.Value = 16#0; SDO List.Clear pdo mapping.Size = 8; SDO List.Clear pdo mapping.AbortIfError = FALSE; SDO List.Clear pdo mapping.JumpToLine = FALSE; SDO List.Clear pdo mapping.Line = 0; SDO List.Set Mapping.Index = 16#1A02; SDO List.Set Mapping.Subindex = 16#01; SDO List.Set Mapping.Value = 16#32010008; SDO List.Set Mapping.Size = 32; SDO List.Set Mapping.AbortIfError = FALSE; SDO List.Set Mapping.JumpToLine = FALSE; SDO List.Set Mapping.Line = 0; SDO List.Set Mapping.Index = 16#1A02; SDO List.Set Mapping.Subindex = 16#02; SDO List.Set Mapping.Value = 16#32020008; SDO List.Set Mapping.Size = 32; SDO List.Set Mapping.AbortIfError = FALSE; SDO List.Set Mapping.JumpToLine = FALSE; SDO List.Set Mapping.Line = 0; SDO List.Set Mapping.Index = 16#1A02;
              SDO List.Set Mapping.Subindex = 16#03; SDO List.Set Mapping.Value = 16#32030008; SDO List.Set Mapping.Size = 32; SDO List.Set Mapping.AbortIfError = FALSE; SDO List.Set Mapping.JumpToLine = FALSE; SDO List.Set Mapping.Line = 0; SDO List.Set Mapping.Index = 16#1A02; SDO List.Set Mapping.Subindex = 16#04; SDO List.Set Mapping.Value = 16#32040008; SDO List.Set Mapping.Size = 32; SDO List.Set Mapping.AbortIfError = FALSE; SDO List.Set Mapping.JumpToLine = FALSE; SDO List.Set Mapping.Line = 0; SDO List.Set Mapping.Index = 16#1A02; SDO List.Set Mapping.Subindex = 16#05; SDO List.Set Mapping.Value = 16#32050008; SDO List.Set Mapping.Size = 32; SDO List.Set Mapping.AbortIfError = FALSE; SDO List.Set Mapping.JumpToLine = FALSE; SDO List.Set Mapping.Line = 0; SDO List.Set Mapping.Index = 16#1A02; SDO List.Set Mapping.Subindex = 16#06; SDO List.Set Mapping.Value = 16#32060008; SDO List.Set Mapping.Size = 32; SDO List.Set Mapping.AbortIfError = FALSE; SDO List.Set Mapping.JumpToLine = FALSE; SDO List.Set Mapping.Line = 0; SDO List.Set Mapping.Index = 16#1A02; SDO List.Set Mapping.Subindex = 16#07; SDO List.Set Mapping.Value = 16#32070008; SDO List.Set Mapping.Size = 32; SDO List.Set Mapping.AbortIfError = FALSE; SDO List.Set Mapping.JumpToLine = FALSE; SDO List.Set Mapping.Line = 0; SDO List.Set Mapping.Index = 16#1A02; SDO List.Set Mapping.Subindex = 16#08; SDO List.Set Mapping.Value = 16#32080008; SDO List.Set Mapping.Size = 32; SDO List.Set Mapping.AbortIfError = FALSE; SDO List.Set Mapping.JumpToLine = FALSE;
              SDO List.Set Mapping.Line = 0; SDO List.Set number of mappings.Index = 16#1A02; SDO List.Set number of mappings.Subindex = 16#00; SDO List.Set number of mappings.Value = 16#08; SDO List.Set number of mappings.Size = 8; SDO List.Set number of mappings.AbortIfError = FALSE; SDO List.Set number of mappings.JumpToLine = FALSE; SDO List.Set number of mappings.Line = 0; SDO List.Set and enable COB-ID.Index = 16#1802; SDO List.Set and enable COB-ID.Subindex = 16#01; SDO List.Set and enable COB-ID.Value = 16#00000382; SDO List.Set and enable COB-ID.Size = 32; SDO List.Set and enable COB-ID.AbortIfError = FALSE; SDO List.Set and enable COB-ID.JumpToLine = FALSE; SDO List.Set and enable COB-ID.Line = 0; SDO List.Disable PDO.Index = 16#1803; SDO List.Disable PDO.Subindex = 16#01; SDO List.Disable PDO.Value = 16#80000482; SDO List.Disable PDO.Size = 32; SDO List.Disable PDO.AbortIfError = FALSE; SDO List.Disable PDO.JumpToLine = FALSE; SDO List.Disable PDO.Line = 0; SDO List.Set transmission type.Index = 16#1803; SDO List.Set transmission type.Subindex = 16#02; SDO List.Set transmission type.Value = 16#FF; SDO List.Set transmission type.Size = 8; SDO List.Set transmission type.AbortIfError = FALSE; SDO List.Set transmission type.JumpToLine = FALSE; SDO List.Set transmission type.Line = 0; SDO List.Set inhibit time.Index = 16#1803; SDO List.Set inhibit time.Subindex = 16#03; SDO List.Set inhibit time.Value = 16#0000; SDO List.Set inhibit time.Size = 16; SDO List.Set inhibit time.AbortIfError = FALSE; SDO List.Set inhibit time.JumpToLine = FALSE; SDO List.Set inhibit time.Line = 0; SDO List.Clear pdo mapping.Index = 16#1A03; SDO List.Clear pdo mapping.Subindex = 16#00; SDO List.Clear pdo mapping.Value = 16#0; SDO List.Clear pdo mapping.Size = 8;
              SDO List.Clear pdo mapping.AbortIfError = FALSE; SDO List.Clear pdo mapping.JumpToLine = FALSE; SDO List.Clear pdo mapping.Line = 0; SDO List.Set Mapping.Index = 16#1A03; SDO List.Set Mapping.Subindex = 16#01; SDO List.Set Mapping.Value = 16#32090008; SDO List.Set Mapping.Size = 32; SDO List.Set Mapping.AbortIfError = FALSE; SDO List.Set Mapping.JumpToLine = FALSE; SDO List.Set Mapping.Line = 0; SDO List.Set Mapping.Index = 16#1A03; SDO List.Set Mapping.Subindex = 16#02; SDO List.Set Mapping.Value = 16#32100008; SDO List.Set Mapping.Size = 32; SDO List.Set Mapping.AbortIfError = FALSE; SDO List.Set Mapping.JumpToLine = FALSE; SDO List.Set Mapping.Line = 0; SDO List.Set Mapping.Index = 16#1A03; SDO List.Set Mapping.Subindex = 16#03; SDO List.Set Mapping.Value = 16#32110008; SDO List.Set Mapping.Size = 32; SDO List.Set Mapping.AbortIfError = FALSE; SDO List.Set Mapping.JumpToLine = FALSE; SDO List.Set Mapping.Line = 0; SDO List.Set Mapping.Index = 16#1A03; SDO List.Set Mapping.Subindex = 16#04; SDO List.Set Mapping.Value = 16#32120008; SDO List.Set Mapping.Size = 32; SDO List.Set Mapping.AbortIfError = FALSE; SDO List.Set Mapping.JumpToLine = FALSE; SDO List.Set Mapping.Line = 0; SDO List.Set Mapping.Index = 16#1A03; SDO List.Set Mapping.Subindex = 16#05; SDO List.Set Mapping.Value = 16#32130008; SDO List.Set Mapping.Size = 32; SDO List.Set Mapping.AbortIfError = FALSE; SDO List.Set Mapping.JumpToLine = FALSE; SDO List.Set Mapping.Line = 0; SDO List.Set Mapping.Index = 16#1A03; SDO List.Set Mapping.Subindex = 16#06;
              SDO List.Set Mapping.Value = 16#32140008; SDO List.Set Mapping.Size = 32; SDO List.Set Mapping.AbortIfError = FALSE; SDO List.Set Mapping.JumpToLine = FALSE; SDO List.Set Mapping.Line = 0; SDO List.Set Mapping.Index = 16#1A03; SDO List.Set Mapping.Subindex = 16#07; SDO List.Set Mapping.Value = 16#32150008; SDO List.Set Mapping.Size = 32; SDO List.Set Mapping.AbortIfError = FALSE; SDO List.Set Mapping.JumpToLine = FALSE; SDO List.Set Mapping.Line = 0; SDO List.Set Mapping.Index = 16#1A03; SDO List.Set Mapping.Subindex = 16#08; SDO List.Set Mapping.Value = 16#32160008; SDO List.Set Mapping.Size = 32; SDO List.Set Mapping.AbortIfError = FALSE; SDO List.Set Mapping.JumpToLine = FALSE; SDO List.Set Mapping.Line = 0; SDO List.Set number of mappings.Index = 16#1A03; SDO List.Set number of mappings.Subindex = 16#00; SDO List.Set number of mappings.Value = 16#08; SDO List.Set number of mappings.Size = 8; SDO List.Set number of mappings.AbortIfError = FALSE; SDO List.Set number of mappings.JumpToLine = FALSE; SDO List.Set number of mappings.Line = 0; SDO List.Set and enable COB-ID.Index = 16#1803; SDO List.Set and enable COB-ID.Subindex = 16#01; SDO List.Set and enable COB-ID.Value = 16#00000482; SDO List.Set and enable COB-ID.Size = 32; SDO List.Set and enable COB-ID.AbortIfError = FALSE; SDO List.Set and enable COB-ID.JumpToLine = FALSE; SDO List.Set and enable COB-ID.Line = 0; ConfigVersion = 50659584
            unmapped channels: CCON, CPOS, REC_NR/CDIR, RES/DEM_VAL1/PARA1, RES/DEM_VAL2/PARA2, RES, SUBINDEX, REQCODE_PNU, PARAVAL, FHPP+_O_Byte01, FHPP+_O_Byte02, FHPP+_O_Byte03, FHPP+_O_Byte04, FHPP+_O_Byte05, FHPP+_O_Byte06, FHPP+_O_Byte07, FHPP+_O_Byte08, FHPP+_O_Byte09, FHPP+_O_Byte10, FHPP+_O_Byte11, FHPP+_O_Byte12, FHPP+_O_Byte13, FHPP+_O_Byte14, FHPP+_O_Byte15, FHPP+_O_Byte16, SCON, SPOS, REC_NR/SDIR, RSB/ACT_VAL1, ACT_POS/ACT_VAL2, RES, SUBINDEX, RESPCODE_PNU, PARAVAL, FHPP+_I_Byte01, FHPP+_I_Byte02, FHPP+_I_Byte03, FHPP+_I_Byte04, FHPP+_I_Byte05, FHPP+_I_Byte06,
              FHPP+_I_Byte07, FHPP+_I_Byte08, FHPP+_I_Byte09, FHPP+_I_Byte10, FHPP+_I_Byte11, FHPP+_I_Byte12, FHPP+_I_Byte13, FHPP+_I_Byte14, FHPP+_I_Byte15, FHPP+_I_Byte16
  text list GlobalTextList
*)

// Device/Application/Global
VAR_GLOBAL
	fb_AxisU1Control: FHPP_CTRL;	
	fb_AxisU1Control_Read: FML_Read;
	fb_AxisU1Control_Write: FML_Write;
	
	fb_AxisU2Control: FHPP_CTRL;	
	fb_AxisU2Control_Read: FML_Read;
	fb_AxisU2Control_Write: FML_Write;
	
	fb_AxisU3Control: FHPP_CTRL;	
	fb_AxisU3Control_Read: FML_Read;
	fb_AxisU3Control_Write: FML_Write;
	
	Data_Ref_U1: DT_FML_REF;
	Data_Ref_U2: DT_FML_REF;
	Data_Ref_U3: DT_FML_REF;
	Input_U1 AT %IB4: ARRAY [0..7] OF BYTE;
	Output_U1 AT %QB4: ARRAY [0..7] OF BYTE;
	Input_U2 AT %IB36: ARRAY [0..7] OF BYTE;
	Output_U2 AT %QB36: ARRAY [0..7] OF BYTE;
	Input_U3 AT %IB68: ARRAY [0..7] OF BYTE;
	Output_U3 AT %QB68: ARRAY [0..7] OF BYTE;
	
	
	g_iCaseOtoPrg: INT;

	DI_StartButton  AT %IX1.1: BOOL;
	tonWaitU1: Ton;
	g_bStartaBasildi: BOOL;
	DI_Stop AT %ix1.2: BOOL;
END_VAR

// Device/Application/Main_PRG
PROGRAM Main_PRG
VAR
END_VAR

Fhpp();
Motion_PRG();

END_PROGRAM

// Device/Application/FHPP
PROGRAM FHPP
VAR
	
	
END_VAR

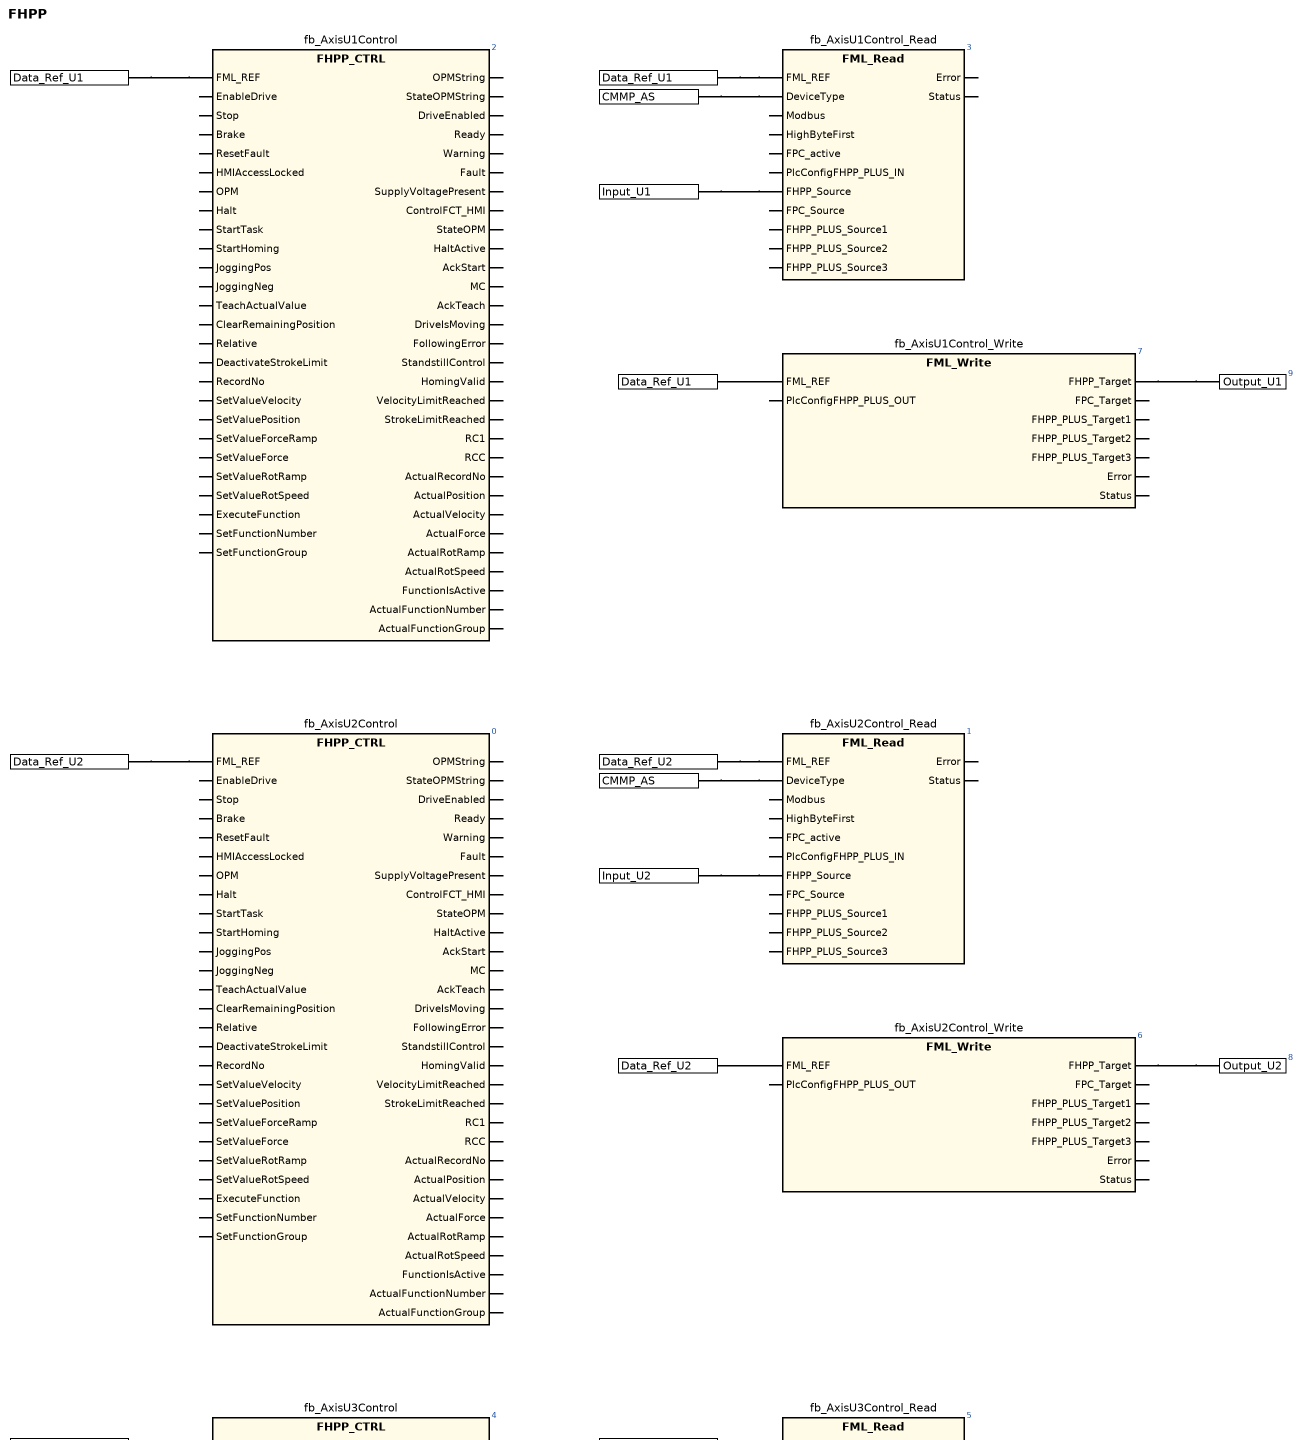
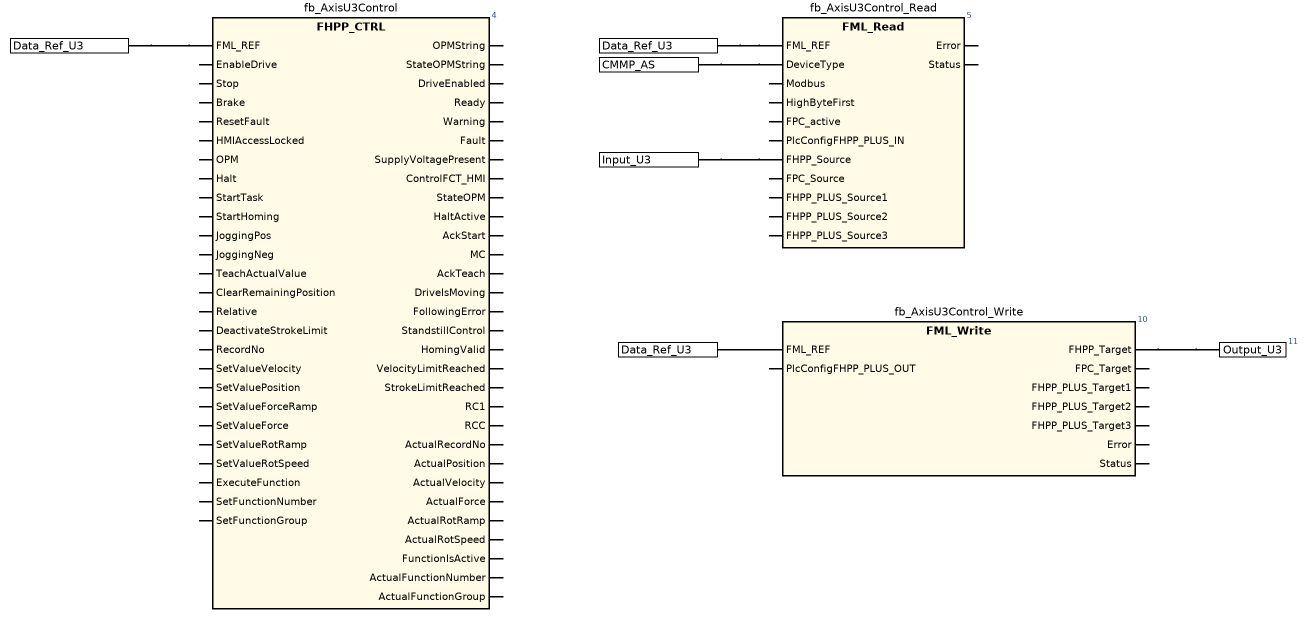
fb_AxisU2Control(FML_REF := Data_Ref_U2); // FHPP_CTRL
fb_AxisU2Control_Read(FML_REF := Data_Ref_U2, DeviceType := CMMP_AS, FHPP_Source := Input_U2); // FML_Read
fb_AxisU1Control(FML_REF := Data_Ref_U1); // FHPP_CTRL
fb_AxisU1Control_Read(FML_REF := Data_Ref_U1, DeviceType := CMMP_AS, FHPP_Source := Input_U1); // FML_Read
fb_AxisU3Control(FML_REF := Data_Ref_U3); // FHPP_CTRL
fb_AxisU3Control_Read(FML_REF := Data_Ref_U3, DeviceType := CMMP_AS, FHPP_Source := Input_U3); // FML_Read
fb_AxisU2Control_Write(FML_REF := Data_Ref_U2); // FML_Write
fb_AxisU1Control_Write(FML_REF := Data_Ref_U1); // FML_Write
Output_U2 := fb_AxisU2Control_Write.FHPP_Target;
Output_U1 := fb_AxisU1Control_Write.FHPP_Target;
fb_AxisU3Control_Write(FML_REF := Data_Ref_U3); // FML_Write
Output_U3 := fb_AxisU3Control_Write.FHPP_Target;

END_PROGRAM

// Device/Application/Motion_PRG
PROGRAM Motion_PRG
VAR
	R_TrigU1Fault: R_Trig;
	TonReset: Ton;
END_VAR

CASE g_iCaseOtoPrg OF
	
0:
IF DI_StartButton THEN
	g_bStartaBasildi :=TRUE;
	g_iCaseOtoPrg := 1;	
END_IF

1:
	fb_AxisU1Control.EnableDrive	:=FALSE;
	fb_AxisU1Control.Stop			:=FALSE;
	fb_AxisU1Control.Brake			:=FALSE;
	fb_AxisU1Control.Halt			:=FALSE;
	fb_AxisU1Control.ResetFault		:=FALSE;
	fb_AxisU1Control.StartHoming	:=FALSE;
	fb_AxisU1Control.StartTask		:=FALSE;
	fb_AxisU1Control.JoggingNeg		:=FALSE;
	fb_AxisU1Control.JoggingPos		:=FALSE;
	
	fb_AxisU2Control.EnableDrive	:=FALSE;
	fb_AxisU2Control.Stop			:=FALSE;
	fb_AxisU2Control.Brake			:=FALSE;
	fb_AxisU2Control.Halt			:=FALSE;
	fb_AxisU2Control.ResetFault		:=FALSE;
	fb_AxisU2Control.StartHoming	:=FALSE;
	fb_AxisU2Control.StartTask		:=FALSE;
	fb_AxisU2Control.JoggingNeg		:=FALSE;
	fb_AxisU2Control.JoggingPos		:=FALSE;
	
	fb_AxisU3Control.EnableDrive	:=FALSE;
	fb_AxisU3Control.Stop			:=FALSE;
	fb_AxisU3Control.Brake			:=FALSE;
	fb_AxisU3Control.Halt			:=FALSE;
	fb_AxisU3Control.ResetFault		:=FALSE;
	fb_AxisU3Control.StartHoming	:=FALSE;
	fb_AxisU3Control.StartTask		:=FALSE;
	fb_AxisU3Control.JoggingNeg		:=FALSE;
	fb_AxisU3Control.JoggingPos		:=FALSE;
	
	g_iCaseOtoPrg					:= 10;	

10:
IF fb_AxisU1Control.Fault
OR fb_AxisU2Control.Fault
OR fb_AxisU3Control.Fault 
THEN
	fb_AxisU1Control.ResetFault	:=TRUE;
	fb_AxisU2Control.ResetFault	:=TRUE;
	fb_AxisU3Control.ResetFault	:=TRUE;
	g_iCaseOtoPrg				:=20;
ELSE
	g_iCaseOtoPrg				:=20;		
END_IF

20:
tonWaitU1(IN:=TRUE,PT:=T#250MS);
	IF fb_AxisU1Control.SupplyVoltagePresent
	AND	fb_AxisU2Control.SupplyVoltagePresent
	AND	fb_AxisU3Control.SupplyVoltagePresent
	AND tonWaitU1.Q
	THEN
		tonWaitU1(IN:=FALSE);
		fb_AxisU1Control.Halt		:=TRUE;
		fb_AxisU1Control.Stop		:=TRUE;
		fb_AxisU1Control.ResetFault	:=FALSE;
		fb_AxisU2Control.Halt		:=TRUE;
		fb_AxisU2Control.Stop		:=TRUE;
		fb_AxisU2Control.ResetFault	:=FALSE;
		fb_AxisU3Control.Halt		:=TRUE;
		fb_AxisU3Control.Stop		:=TRUE;
		fb_AxisU3Control.ResetFault	:=FALSE;
		g_iCaseOtoPrg				:=30;
	END_IF
	
30:
tonWaitU1(in:=TRUE, pt:=T#100MS);
IF tonWaitU1.q
AND NOT fb_AxisU1Control.Fault	
AND NOT fb_AxisU2Control.Fault
AND NOT fb_AxisU3Control.Fault
THEN
	tonWaitU1(in:=FALSE);
	fb_AxisU1Control.EnableDrive	:=TRUE;
	fb_AxisU2Control.EnableDrive	:=TRUE;
	fb_AxisU3Control.EnableDrive	:=TRUE;
	g_iCaseOtoPrg					:=40;
ELSIF tonWaitU1.q
AND fb_AxisU1Control.Fault
OR fb_AxisU2Control.Fault
OR fb_AxisU3Control.Fault
THEN
	tonWaitU1(in:=FALSE);
	g_iCaseOtoPrg					:=10;	
END_IF

40:
tonWaitU1(in:=NOT fb_AxisU1Control.DriveEnabled
OR NOT fb_AxisU2Control.DriveEnabled
OR NOT fb_AxisU3Control.DriveEnabled,
pt:=T#1S);
	IF tonWaitU1.Q
	THEN
		g_iCaseOtoPrg					:=10;
	END_IF
	
	IF fb_AxisU1Control.DriveEnabled
		AND fb_AxisU2Control.DriveEnabled
		AND fb_AxisU3Control.DriveEnabled
	THEN
		g_iCaseOtoPrg					:=50;	
	END_IF

50:
(*Z Servo U3 Referans Yapacak*)
	tonWaitU1(in:=TRUE, pt:=T#250MS);
	IF NOT fb_AxisU3Control.HomingValid
	AND tonWaitU1.Q
	THEN
		fb_AxisU3Control.StartHoming := TRUE;
		tonWaitU1(in:=FALSE);
		g_iCaseOtoPrg 				 := 60;	
	ELSIF fb_AxisU3Control.HomingValid
	AND tonWaitU1.Q
	THEN
		tonWaitU1(in:=FALSE);
		g_iCaseOtoPrg 				 := 51;			
	END_IF

60:
	IF NOT fb_AxisU3Control.HomingValid
	AND NOT fb_AxisU3Control.MC
	THEN
		g_iCaseOtoPrg := 70;
	ELSIF fb_AxisU3Control.MC
	THEN
		fb_AxisU3Control.StartHoming := FALSE;	
		g_iCaseOtoPrg 				 := 50;			
	END_IF

70:
	IF fb_AxisU3Control.HomingValid
	THEN
		fb_AxisU3Control.StartHoming 	:= FALSE;
		g_iCaseOtoPrg 					:= 51;
	END_IF

51:
(*X ve Y Servo U1-2 Referans Yapacak*)

tonWaitU1(in:=TRUE, pt:=T#250MS);
	IF tonWaitU1.Q
	AND( NOT fb_AxisU1Control.HomingValid 
		OR NOT fb_AxisU2Control.HomingValid )
	THEN
		fb_AxisU1Control.StartHoming := TRUE;
		fb_AxisU2Control.StartHoming := TRUE;
		tonWaitU1(in:=FALSE);
		g_iCaseOtoPrg 				 := 61;	
	ELSIF fb_AxisU1Control.HomingValid 
	AND fb_AxisU2Control.HomingValid
	AND tonWaitU1.Q
	THEN
		tonWaitU1(in:=FALSE);
		g_iCaseOtoPrg 				 := 80;			
	END_IF

61:
	IF (NOT fb_AxisU1Control.HomingValid
	AND NOT fb_AxisU1Control.MC)
	OR (NOT fb_AxisU2Control.HomingValid
	AND NOT fb_AxisU2Control.MC)
	THEN
		g_iCaseOtoPrg := 71;
	ELSIF fb_AxisU1Control.MC
		AND fb_AxisU2Control.MC
	THEN
		fb_AxisU1Control.StartHoming := FALSE;
		fb_AxisU2Control.StartHoming := FALSE;		
		g_iCaseOtoPrg 				 := 51;			
	END_IF

71:
	IF fb_AxisU1Control.HomingValid
	AND fb_AxisU2Control.HomingValid
	THEN
		fb_AxisU3Control.StartHoming 	:= FALSE;
		fb_AxisU2Control.StartHoming 	:= FALSE;	
		g_iCaseOtoPrg 					:= 51;
	END_IF
	
	
	(* X ekseni birinci hareket*)
80:
IF fb_AxisU1Control.DriveEnabled
	AND fb_AxisU1Control.Ready
	AND DI_stop
	THEN
		g_iCaseOtoPrg 					:= 90;
	END_IF

90:
	fb_AxisU1Control.OPM				:=1;
	fb_AxisU1Control.SetValueVelocity	:=50;
	fb_AxisU1Control.SetValuePosition	:=70000;
	fb_AxisU1Control.StartTask			:=TRUE;
	g_iCaseOtoPrg 						:=100;

100:
tonWaitU1(in:=TRUE, pt:=T#100MS);
IF tonWaitU1.Q AND fb_AxisU1Control.AckStart
	AND (fb_AxisU1Control.DriveIsMoving OR NOT fb_AxisU1Control.MC)
	THEN
		fb_AxisU1Control.StartTask		:=FALSE;
		tonWaitU1(IN:=FALSE);
		g_iCaseOtoPrg 					:=110;
	END_IF

110:
	IF NOT fb_AxisU1Control.DriveIsMoving
	AND fb_AxisU1Control.MC
	THEN
		fb_AxisU1Control.StartTask		:=FALSE;
		g_iCaseOtoPrg 					:=81;
	END_IF

	
	(* Y ekseni birinci hareket*)
81:
IF fb_AxisU2Control.DriveEnabled
	AND fb_AxisU2Control.Ready
	AND DI_stop
	THEN
		g_iCaseOtoPrg 					:= 91;
	END_IF

91:
	fb_AxisU2Control.OPM				:=1;
	fb_AxisU2Control.SetValueVelocity	:=50;
	fb_AxisU2Control.SetValuePosition	:=50000;
	fb_AxisU2Control.StartTask			:=TRUE;
	g_iCaseOtoPrg 						:=101;

101:
tonWaitU1(in:=TRUE, pt:=T#100MS);
IF tonWaitU1.q AND fb_AxisU2Control.AckStart
	AND (fb_AxisU2Control.DriveIsMoving OR NOT fb_AxisU2Control.MC)
	THEN
		fb_AxisU2Control.StartTask		:=FALSE;
		tonWaitU1(IN:=FALSE);
		g_iCaseOtoPrg 					:=111;
	END_IF

111:
	IF NOT fb_AxisU2Control.DriveIsMoving
	AND fb_AxisU2Control.MC
	THEN
		fb_AxisU2Control.StartTask		:=FALSE;
		g_iCaseOtoPrg 					:=82;
	END_IF


	(* Z ekseni birinci hareket*)
82:
IF fb_AxisU3Control.DriveEnabled
	AND fb_AxisU3Control.Ready
	AND DI_stop
	THEN
		g_iCaseOtoPrg 					:= 92;
	END_IF

92:
	fb_AxisU3Control.OPM				:=1;
	fb_AxisU3Control.SetValueVelocity	:=50;
	fb_AxisU3Control.SetValuePosition	:=90000;
	fb_AxisU3Control.StartTask			:=TRUE;
	g_iCaseOtoPrg 						:=102;

102:
tonWaitU1(in:=TRUE, pt:=T#100MS);
IF tonWaitU1.Q AND fb_AxisU3Control.AckStart
	AND (fb_AxisU3Control.DriveIsMoving OR NOT fb_AxisU3Control.MC)
	THEN
		fb_AxisU3Control.StartTask		:=FALSE;
		tonWaitU1(IN:=FALSE);
		g_iCaseOtoPrg 					:=112;
	END_IF

112:
	IF NOT fb_AxisU3Control.DriveIsMoving
	AND fb_AxisU3Control.MC
	THEN
		fb_AxisU3Control.StartTask		:=FALSE;
		g_iCaseOtoPrg 					:=83;
	END_IF

	(* X ekseni 2. hareket*)
83:
IF fb_AxisU1Control.DriveEnabled
	AND fb_AxisU1Control.Ready
	AND DI_stop
	THEN
		g_iCaseOtoPrg 					:= 93;
	END_IF

93:
	fb_AxisU1Control.OPM				:=1;
	fb_AxisU1Control.SetValueVelocity	:=80;
	fb_AxisU1Control.SetValuePosition	:=170000;
	fb_AxisU1Control.StartTask			:=TRUE;
	g_iCaseOtoPrg 						:=103;

103:
tonWaitU1(in:=TRUE, pt:=T#100MS);
IF tonWaitU1.Q AND fb_AxisU1Control.AckStart
	AND (fb_AxisU1Control.DriveIsMoving OR NOT fb_AxisU1Control.MC)
	THEN
		fb_AxisU1Control.StartTask		:=FALSE;
		tonWaitU1(IN:=FALSE);
		g_iCaseOtoPrg 					:=113;
	END_IF

113:
	IF NOT fb_AxisU1Control.DriveIsMoving
	AND fb_AxisU1Control.MC
	THEN
		fb_AxisU1Control.StartTask		:=FALSE;
		g_iCaseOtoPrg 					:=84;
	END_IF

	(* Y ekseni 2. hareket*)
84:
IF fb_AxisU2Control.DriveEnabled 
	AND fb_AxisU2Control.Ready
	AND DI_stop
	THEN
		g_iCaseOtoPrg 					:= 94;
	END_IF

94:
	fb_AxisU2Control.OPM				:=1;
	fb_AxisU2Control.SetValueVelocity	:=70;
	fb_AxisU2Control.SetValuePosition	:=230000;
	fb_AxisU2Control.StartTask			:=TRUE;
	g_iCaseOtoPrg 						:=104;

104:
tonWaitU1(in:=TRUE, pt:=T#100MS);
IF tonWaitU1.Q AND fb_AxisU2Control.AckStart
	AND (fb_AxisU2Control.DriveIsMoving OR NOT fb_AxisU2Control.MC)
	THEN
		fb_AxisU2Control.StartTask		:=FALSE;
		tonWaitU1(IN:=FALSE);
		g_iCaseOtoPrg 					:=114;
	END_IF

114:
	IF NOT fb_AxisU2Control.DriveIsMoving
	AND fb_AxisU2Control.MC
	THEN
		fb_AxisU2Control.StartTask		:=FALSE;
		g_iCaseOtoPrg 					:=85;
	END_IF
	
	
		(* Z ekseni 2. hareket*)
85:
IF fb_AxisU3Control.DriveEnabled
	AND fb_AxisU3Control.Ready
	AND DI_stop
	THEN
		g_iCaseOtoPrg 					:= 95;
	END_IF

95:
	fb_AxisU3Control.OPM				:=1;
	fb_AxisU3Control.SetValueVelocity	:=50;
	fb_AxisU3Control.SetValuePosition	:=160000;
	fb_AxisU3Control.StartTask			:=TRUE;
	g_iCaseOtoPrg 						:=105;

105:
tonWaitU1(in:=TRUE, pt:=T#100MS);
IF tonWaitU1.Q AND fb_AxisU3Control.AckStart
	AND (fb_AxisU3Control.DriveIsMoving OR NOT fb_AxisU3Control.MC)
	THEN
		fb_AxisU3Control.StartTask		:=FALSE;
		tonWaitU1(IN:=FALSE);
		g_iCaseOtoPrg 					:=115;
	END_IF

115:
	IF NOT fb_AxisU3Control.DriveIsMoving
	AND fb_AxisU3Control.MC
	THEN
		fb_AxisU3Control.StartTask		:=FALSE;
		g_iCaseOtoPrg 					:=80;
	END_IF
	
END_CASE


TonReset(IN:= Not DI_Stop, PT:= T#3S);
IF TonReset.Q THEN
	fb_AxisU1Control.ResetFault	:= TRUE;
	TonReset(IN:=FALSE);
	g_iCaseOtoPrg 				:=0;
END_IF

END_PROGRAM

// Device/Application/PO3_Axis/AxisX/PrgAxisXCallPrg
PROGRAM PrgAxisXCallPrg
VAR
END_VAR

;

END_PROGRAM

// Device/Application/Visualization
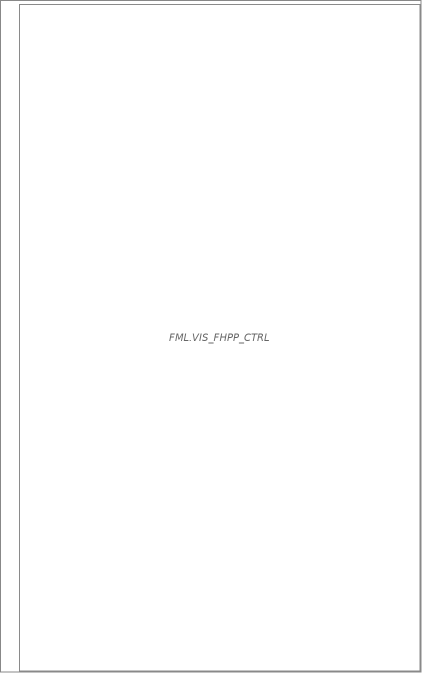
VISUALIZATION Visualization  // 422x673
    Frame (19,4 401x667)
        shows FML.VIS_FHPP_CTRL(m_Input_INST := fb_AxisU1Control)
END_VISUALIZATION
